C05472=1200.929,400.993,-81.846,-175.880,8.483,148.485
C05473=1200.932,400.745,-81.811,-175.880,8.481,148.484
C05474=1200.937,400.499,-81.776,-175.881,8.479,148.484
C05475=1200.941,400.250,-81.741,-175.881,8.476,148.483
C05476=1200.944,400.003,-81.706,-175.882,8.474,148.483
C05477=1200.949,399.756,-81.671,-175.882,8.471,148.482
C05478=1200.953,399.508,-81.636,-175.883,8.469,148.482
C05479=1200.957,399.261,-81.601,-175.883,8.466,148.481
C05480=1200.961,399.013,-81.566,-175.884,8.464,148.480
C05481=1200.965,398.766,-81.532,-175.884,8.462,148.480
C05482=1200.968,398.519,-81.496,-175.885,8.458,148.479
C05483=1200.972,398.270,-81.461,-175.885,8.456,148.479
C05484=1200.977,398.024,-81.426,-175.885,8.454,148.478
C05485=1200.981,397.775,-81.391,-175.886,8.451,148.478
C05486=1200.985,397.529,-81.356,-175.886,8.449,148.477
C05487=1200.989,397.281,-81.321,-175.887,8.447,148.477
C05488=1200.993,397.033,-81.287,-175.887,8.443,148.476
C05489=1200.997,396.786,-81.251,-175.888,8.441,148.476
C05490=1201.001,396.537,-81.217,-175.888,8.439,148.475
C05491=1201.004,396.291,-81.182,-175.889,8.436,148.475
C05492=1201.008,396.043,-81.147,-175.889,8.434,148.474
C05493=1201.013,395.795,-81.113,-175.890,8.430,148.473
C05494=1201.017,395.548,-81.077,-175.890,8.428,148.473
C05495=1201.021,395.301,-81.043,-175.891,8.426,148.473
C05496=1201.025,395.053,-81.007,-175.891,8.423,148.472
C05497=1201.029,394.806,-80.973,-175.892,8.421,148.471
C05498=1201.033,394.558,-80.938,-175.892,8.418,148.471
C05499=1201.036,394.310,-80.903,-175.893,8.415,148.470
C05500=1201.041,394.063,-80.868,-175.893,8.412,148.470
C05501=1201.045,393.815,-80.834,-175.894,8.410,148.469
C05502=1201.049,393.568,-80.798,-175.895,8.407,148.469
C05503=1201.053,393.320,-80.764,-175.895,8.405,148.468
C05504=1201.057,393.073,-80.730,-175.896,8.402,148.468
C05505=1201.062,392.790,-80.689,-175.896,8.400,148.467
C05506=1201.067,392.507,-80.650,-175.897,8.397,148.467
C05507=1201.070,392.224,-80.610,-175.898,8.393,148.466
C05508=1201.076,391.941,-80.570,-175.898,8.390,148.465
C05509=1201.079,391.694,-80.536,-175.899,8.387,148.465
C05510=1201.083,391.446,-80.501,-175.899,8.385,148.464
C05511=1201.088,391.199,-80.466,-175.900,8.382,148.464
C05512=1201.091,390.951,-80.431,-175.900,8.380,148.463
C05513=1201.096,390.704,-80.396,-175.901,8.376,148.463
C05514=1201.099,390.456,-80.362,-175.902,8.374,148.462
C05515=1201.104,390.209,-80.328,-175.903,8.371,148.462
C05516=1201.107,389.961,-80.292,-175.903,8.368,148.461
C05517=1201.112,389.714,-80.258,-175.904,8.365,148.460
C05518=1201.115,389.466,-80.223,-175.904,8.363,148.460
C05519=1201.120,389.218,-80.189,-175.906,8.360,148.460
C05520=1201.124,388.970,-80.154,-175.906,8.357,148.459
C05521=1201.128,388.724,-80.119,-175.907,8.355,148.458
C05522=1201.131,388.476,-80.085,-175.907,8.352,148.458
C05523=1201.136,388.228,-80.050,-175.909,8.349,148.457
C05524=1201.140,387.980,-80.015,-175.909,8.347,148.457
C05525=1201.144,387.733,-79.981,-175.910,8.343,148.456
C05526=1201.147,387.486,-79.946,-175.910,8.340,148.456
C05527=1201.152,387.238,-79.912,-175.911,8.338,148.455
C05528=1201.156,386.990,-79.877,-175.912,8.335,148.455
C05529=1201.160,386.743,-79.843,-175.913,8.332,148.454
C05530=1201.164,386.495,-79.808,-175.914,8.329,148.454
C05531=1201.168,386.247,-79.774,-175.915,8.326,148.453
C05532=1201.172,386.000,-79.740,-175.915,8.324,148.453
C05533=1201.176,385.752,-79.705,-175.916,8.321,148.452
C05534=1201.180,385.505,-79.670,-175.917,8.318,148.452
C05535=1201.184,385.257,-79.635,-175.918,8.315,148.451
C05536=1201.188,385.010,-79.601,-175.919,8.312,148.451
C05537=1201.192,384.762,-79.566,-175.920,8.309,148.450
C05538=1201.197,384.515,-79.532,-175.920,8.307,148.450
C05539=1201.200,384.267,-79.497,-175.921,8.304,148.449
C05540=1201.204,384.019,-79.463,-175.922,8.301,148.449
C05541=1201.209,383.772,-79.428,-175.923,8.298,148.448
C05542=1201.212,383.524,-79.394,-175.924,8.295,148.448
C05543=1201.217,383.277,-79.360,-175.925,8.292,148.447
C05544=1201.220,383.029,-79.326,-175.926,8.289,148.447
C05545=1201.225,382.781,-79.291,-175.927,8.286,148.446
C05546=1201.228,382.533,-79.256,-175.927,8.283,148.445
C05547=1201.232,382.286,-79.222,-175.928,8.280,148.445
C05548=1201.237,382.039,-79.188,-175.929,8.277,148.444
C05549=1201.241,381.791,-79.153,-175.930,8.275,148.444
C05550=1201.245,381.544,-79.119,-175.931,8.272,148.444
C05551=1201.249,381.295,-79.084,-175.932,8.269,148.443
C05552=1201.252,381.048,-79.051,-175.933,8.266,148.443
C05553=1201.257,380.801,-79.016,-175.934,8.263,148.442
C05554=1201.261,380.553,-78.981,-175.935,8.260,148.442
C05555=1201.265,380.306,-78.947,-175.936,8.257,148.441
C05556=1201.269,380.058,-78.913,-175.937,8.253,148.441
C05557=1201.273,379.810,-78.879,-175.938,8.251,148.440
C05558=1201.277,379.563,-78.844,-175.940,8.248,148.440
C05559=1201.281,379.315,-78.811,-175.940,8.245,148.439
C05560=1201.285,379.067,-78.776,-175.942,8.242,148.439
C05561=1201.289,378.820,-78.742,-175.942,8.239,148.438
C05562=1201.293,378.572,-78.707,-175.944,8.236,148.438
C05563=1201.298,378.325,-78.673,-175.944,8.233,148.437
C05564=1201.302,378.077,-78.639,-175.946,8.230,148.437
C05565=1201.305,377.829,-78.604,-175.947,8.227,148.436
C05566=1201.310,377.582,-78.571,-175.948,8.224,148.436
C05567=1201.314,377.334,-78.537,-175.949,8.221,148.435
C05568=1201.317,377.086,-78.502,-175.951,8.218,148.435
C05569=1201.322,376.839,-78.468,-175.951,8.215,148.434
C05570=1201.325,376.591,-78.434,-175.953,8.212,148.434
C05571=1201.330,376.343,-78.400,-175.954,8.209,148.434
C05572=1201.334,376.096,-78.366,-175.955,8.206,148.433
C05573=1201.338,375.848,-78.331,-175.956,8.203,148.433
C05574=1201.342,375.601,-78.297,-175.958,8.199,148.432
C05575=1201.346,375.354,-78.264,-175.959,8.197,148.432
C05576=1201.350,375.106,-78.230,-175.960,8.193,148.431
C05577=1201.354,374.858,-78.196,-175.961,8.191,148.431
C05578=1201.358,374.610,-78.161,-175.962,8.188,148.430
C05579=1201.362,374.363,-78.128,-175.964,8.184,148.430
C05580=1201.366,374.115,-78.093,-175.965,8.181,148.430
C05581=1201.370,373.867,-78.059,-175.966,8.178,148.429
C05582=1201.375,373.620,-78.025,-175.967,8.175,148.429
C05583=1201.378,373.372,-77.991,-175.969,8.172,148.428
C05584=1201.382,373.124,-77.957,-175.970,8.169,148.428
C05585=1201.387,372.877,-77.923,-175.971,8.166,148.427
C05586=1201.390,372.629,-77.889,-175.973,8.163,148.427
C05587=1201.395,372.381,-77.855,-175.974,8.160,148.427
C05588=1201.399,372.133,-77.822,-175.975,8.157,148.426
C05589=1201.403,371.886,-77.788,-175.976,8.154,148.426
C05590=1201.407,371.638,-77.753,-175.978,8.150,148.425
C05591=1201.411,371.391,-77.720,-175.979,8.147,148.425
C05592=1201.415,371.143,-77.686,-175.980,8.145,148.424
C05593=1201.420,370.895,-77.652,-175.982,8.141,148.424
C05594=1201.423,370.648,-77.618,-175.983,8.138,148.424
C05595=1201.427,370.400,-77.584,-175.985,8.135,148.423
C05596=1201.432,370.152,-77.550,-175.986,8.132,148.423
C05597=1201.435,369.905,-77.517,-175.988,8.129,148.422
C05598=1201.439,369.657,-77.483,-175.989,8.125,148.422
C05599=1201.443,369.409,-77.449,-175.991,8.122,148.422
C05600=1201.448,369.162,-77.415,-175.992,8.120,148.421
C05601=1201.451,368.915,-77.382,-175.994,8.116,148.421
C05602=1201.456,368.666,-77.347,-175.995,8.113,148.420
C05603=1201.460,368.419,-77.314,-175.997,8.110,148.420
C05604=1201.464,368.171,-77.280,-175.998,8.107,148.420
C05605=1201.468,367.924,-77.246,-175.999,8.104,148.419
C05606=1201.472,367.676,-77.213,-176.001,8.101,148.419
C05607=1201.476,367.427,-77.179,-176.002,8.098,148.419
C05608=1201.480,367.180,-77.145,-176.004,8.094,148.418
C05609=1201.485,366.900,-77.107,-176.006,8.091,148.418
C05610=1201.490,366.618,-77.069,-176.007,8.088,148.417
C05611=1201.494,366.338,-77.031,-176.009,8.084,148.417
C05612=1201.498,366.058,-76.993,-176.011,8.080,148.416
C05613=1201.502,365.810,-76.960,-176.012,8.077,148.416
C05614=1201.507,365.562,-76.925,-176.014,8.074,148.416
C05615=1201.511,365.315,-76.892,-176.016,8.071,148.415
C05616=1201.515,365.067,-76.859,-176.017,8.068,148.415
C05617=1201.519,364.819,-76.825,-176.019,8.064,148.414
C05618=1201.523,364.571,-76.791,-176.020,8.061,148.414
C05619=1201.527,364.324,-76.758,-176.022,8.058,148.414
C05620=1201.531,364.076,-76.724,-176.024,8.055,148.413
C05621=1201.535,363.829,-76.691,-176.025,8.052,148.413
C05622=1201.540,363.581,-76.657,-176.027,8.049,148.413
C05623=1201.543,363.332,-76.624,-176.029,8.046,148.412
C05624=1201.547,363.085,-76.590,-176.030,8.043,148.412
C05625=1201.551,362.838,-76.557,-176.032,8.039,148.412
C05626=1201.555,362.590,-76.524,-176.033,8.037,148.411
C05627=1201.560,362.342,-76.490,-176.035,8.033,148.411
C05628=1201.564,362.095,-76.456,-176.037,8.030,148.411
C05629=1201.568,361.847,-76.423,-176.039,8.027,148.410
C05630=1201.572,361.599,-76.390,-176.041,8.023,148.410
C05631=1201.576,361.351,-76.356,-176.042,8.021,148.410
C05632=1201.580,361.103,-76.323,-176.044,8.017,148.409
C05633=1201.584,360.855,-76.290,-176.046,8.014,148.409
C05634=1201.588,360.608,-76.256,-176.047,8.011,148.409
C05635=1201.592,360.361,-76.223,-176.049,8.007,148.408
C05636=1201.596,360.113,-76.190,-176.051,8.005,148.408
C05637=1201.600,359.865,-76.157,-176.053,8.001,148.408
C05638=1201.604,359.617,-76.123,-176.054,7.999,148.407
C05639=1201.609,359.369,-76.090,-176.056,7.995,148.407
C05640=1201.613,359.122,-76.057,-176.058,7.992,148.407
C05641=1201.618,358.874,-76.023,-176.060,7.989,148.407
C05642=1201.621,358.625,-75.990,-176.062,7.985,148.406
C05643=1201.625,358.378,-75.957,-176.063,7.983,148.406
C05644=1201.629,358.130,-75.924,-176.065,7.979,148.406
C05645=1201.634,357.882,-75.890,-176.067,7.976,148.405
C05646=1201.638,357.634,-75.857,-176.069,7.973,148.405
C05647=1201.642,357.387,-75.824,-176.071,7.970,148.405
C05648=1201.646,357.139,-75.791,-176.073,7.966,148.404
C05649=1201.650,356.891,-75.758,-176.074,7.964,148.404
C05650=1201.654,356.644,-75.725,-176.076,7.960,148.404
C05651=1201.658,356.396,-75.692,-176.078,7.958,148.404
C05652=1201.662,356.148,-75.659,-176.080,7.954,148.403
C05653=1201.666,355.901,-75.626,-176.082,7.951,148.403
C05654=1201.670,355.653,-75.593,-176.084,7.948,148.403
C05655=1201.674,355.405,-75.559,-176.085,7.945,148.402
C05656=1201.678,355.157,-75.526,-176.088,7.941,148.402
C05657=1201.682,354.910,-75.493,-176.089,7.939,148.402
C05658=1201.687,354.661,-75.461,-176.091,7.935,148.402
C05659=1201.691,354.414,-75.428,-176.093,7.932,148.401
C05660=1201.695,354.166,-75.394,-176.095,7.929,148.401
C05661=1201.699,353.918,-75.361,-176.097,7.926,148.401
C05662=1201.703,353.670,-75.328,-176.098,7.923,148.401
C05663=1201.707,353.423,-75.296,-176.101,7.920,148.400
C05664=1201.711,353.175,-75.263,-176.103,7.917,148.400
C05665=1201.715,352.927,-75.230,-176.104,7.914,148.400
C05666=1201.720,352.679,-75.197,-176.106,7.910,148.399
C05667=1201.724,352.432,-75.164,-176.108,7.907,148.399
C05668=1201.728,352.184,-75.130,-176.110,7.905,148.399
C05669=1201.732,351.936,-75.099,-176.112,7.901,148.399
C05670=1201.736,351.688,-75.065,-176.114,7.898,148.398
C05671=1201.740,351.440,-75.032,-176.116,7.895,148.398
C05672=1201.745,351.193,-75.000,-176.118,7.892,148.398
C05673=1201.749,350.945,-74.967,-176.120,7.888,148.398
C05674=1201.753,350.697,-74.934,-176.122,7.886,148.398
C05675=1201.757,350.449,-74.902,-176.124,7.883,148.397
C05676=1201.761,350.201,-74.869,-176.126,7.879,148.397
C05677=1201.765,349.954,-74.836,-176.128,7.876,148.397
C05678=1201.770,349.705,-74.803,-176.130,7.873,148.397
C05679=1201.773,349.458,-74.771,-176.132,7.870,148.396
C05680=1201.777,349.210,-74.738,-176.134,7.867,148.396
C05681=1201.782,348.962,-74.705,-176.136,7.864,148.396
C05682=1201.786,348.714,-74.672,-176.138,7.861,148.396
C05683=1201.790,348.467,-74.641,-176.140,7.858,148.395
C05684=1201.794,348.219,-74.607,-176.142,7.855,148.395
C05685=1201.799,347.971,-74.575,-176.144,7.851,148.395
C05686=1201.803,347.723,-74.542,-176.145,7.849,148.395
C05687=1201.806,347.476,-74.509,-176.148,7.845,148.394
C05688=1201.811,347.227,-74.477,-176.150,7.842,148.394
C05689=1201.815,346.979,-74.444,-176.152,7.839,148.394
C05690=1201.819,346.732,-74.412,-176.154,7.836,148.394
C05691=1201.823,346.484,-74.379,-176.156,7.833,148.394
C05692=1201.828,346.236,-74.347,-176.158,7.830,148.393
C05693=1201.831,345.988,-74.315,-176.160,7.827,148.393
C05694=1201.835,345.740,-74.282,-176.162,7.823,148.393
C05695=1201.840,345.492,-74.249,-176.164,7.821,148.393
C05696=1201.844,345.245,-74.217,-176.166,7.818,148.393
C05697=1201.848,344.997,-74.184,-176.168,7.814,148.392
C05698=1201.852,344.749,-74.152,-176.170,7.812,148.392
C05699=1201.856,344.501,-74.119,-176.172,7.808,148.392
C05700=1201.861,344.253,-74.087,-176.174,7.805,148.392
C05701=1201.865,344.006,-74.055,-176.176,7.803,148.392
C05702=1201.869,343.758,-74.022,-176.179,7.800,148.392
C05703=1201.873,343.510,-73.991,-176.181,7.796,148.391
C05704=1201.877,343.262,-73.957,-176.183,7.794,148.391
C05705=1201.881,343.014,-73.925,-176.185,7.790,148.391
C05706=1201.886,342.766,-73.893,-176.187,7.787,148.391
C05707=1201.890,342.519,-73.860,-176.189,7.785,148.391
C05708=1201.894,342.270,-73.828,-176.191,7.781,148.390
C05709=1201.898,342.022,-73.796,-176.193,7.778,148.390
C05710=1201.902,341.775,-73.765,-176.195,7.775,148.390
C05711=1201.906,341.527,-73.731,-176.197,7.772,148.390
C05712=1201.910,341.279,-73.700,-176.200,7.769,148.390
C05713=1201.915,341.001,-73.663,-176.202,7.766,148.389
C05714=1201.920,340.722,-73.628,-176.204,7.762,148.389
C05715=1201.924,340.443,-73.591,-176.206,7.759,148.389
C05716=1201.929,340.166,-73.555,-176.209,7.756,148.389
C05717=1201.933,339.918,-73.523,-176.211,7.753,148.389
C05718=1201.938,339.669,-73.490,-176.213,7.749,148.389
C05719=1201.942,339.422,-73.459,-176.215,7.747,148.388
C05720=1201.946,339.174,-73.427,-176.217,7.743,148.388
C05721=1201.950,338.926,-73.394,-176.220,7.740,148.388
C05722=1201.954,338.679,-73.362,-176.222,7.738,148.388
C05723=1201.959,338.430,-73.330,-176.224,7.735,148.388
C05724=1201.962,338.182,-73.298,-176.226,7.731,148.388
C05725=1201.967,337.934,-73.266,-176.228,7.729,148.387
C05726=1201.971,337.687,-73.234,-176.231,7.726,148.387
C05727=1201.975,337.439,-73.202,-176.233,7.722,148.387
C05728=1201.979,337.190,-73.170,-176.234,7.720,148.387
C05729=1201.983,336.943,-73.139,-176.237,7.716,148.387
C05730=1201.988,336.695,-73.106,-176.239,7.713,148.387
C05731=1201.992,336.447,-73.074,-176.241,7.711,148.387
C05732=1201.996,336.199,-73.043,-176.243,7.708,148.386
C05733=1202.000,335.951,-73.010,-176.245,7.704,148.386
C05734=1202.004,335.703,-72.978,-176.248,7.701,148.386
C05735=1202.008,335.456,-72.947,-176.250,7.699,148.386
C05736=1202.013,335.207,-72.915,-176.252,7.695,148.386
C05737=1202.016,334.959,-72.883,-176.255,7.692,148.386
C05738=1202.021,334.712,-72.851,-176.256,7.690,148.386
C05739=1202.025,334.463,-72.819,-176.259,7.687,148.385
C05740=1202.029,334.215,-72.787,-176.261,7.683,148.385
C05741=1202.034,333.967,-72.756,-176.263,7.681,148.385
C05742=1202.037,333.719,-72.724,-176.265,7.678,148.385
C05743=1202.042,333.472,-72.692,-176.268,7.675,148.385
C05744=1202.046,333.224,-72.660,-176.269,7.672,148.385
C05745=1202.050,332.976,-72.629,-176.272,7.669,148.385
C05746=1202.054,332.728,-72.597,-176.274,7.666,148.385
C05747=1202.059,332.479,-72.565,-176.276,7.663,148.384
C05748=1202.063,332.232,-72.534,-176.279,7.660,148.384
C05749=1202.067,331.984,-72.502,-176.281,7.657,148.384
C05750=1202.071,331.736,-72.470,-176.283,7.654,148.384
C05751=1202.075,331.489,-72.439,-176.285,7.651,148.384
C05752=1202.080,331.240,-72.407,-176.288,7.648,148.384
C05753=1202.084,330.992,-72.376,-176.290,7.645,148.384
C05754=1202.088,330.744,-72.344,-176.292,7.642,148.384
C05755=1202.092,330.496,-72.313,-176.294,7.639,148.383
C05756=1202.096,330.248,-72.281,-176.297,7.636,148.383
C05757=1202.101,330.001,-72.249,-176.298,7.634,148.383
C05758=1202.105,329.752,-72.218,-176.301,7.631,148.383
C05759=1202.109,329.505,-72.186,-176.303,7.627,148.383
C05760=1202.113,329.257,-72.155,-176.305,7.625,148.383
C05761=1202.117,329.008,-72.123,-176.308,7.622,148.383
C05762=1202.121,328.761,-72.092,-176.310,7.619,148.383
C05763=1202.125,328.513,-72.060,-176.312,7.616,148.383
C05764=1202.130,328.265,-72.029,-176.315,7.613,148.383
C05765=1202.134,328.016,-71.997,-176.317,7.610,148.382
C05766=1202.139,327.768,-71.966,-176.319,7.608,148.382
C05767=1202.142,327.520,-71.934,-176.321,7.604,148.382
C05768=1202.147,327.272,-71.903,-176.324,7.601,148.382
C05769=1202.151,327.024,-71.872,-176.326,7.598,148.382
C05770=1202.155,326.777,-71.840,-176.328,7.596,148.382
C05771=1202.159,326.528,-71.809,-176.331,7.592,148.382
C05772=1202.163,326.281,-71.778,-176.333,7.589,148.382
C05773=1202.167,326.032,-71.746,-176.335,7.587,148.382
C05774=1202.172,325.785,-71.715,-176.338,7.584,148.382
C05775=1202.176,325.537,-71.684,-176.340,7.580,148.381
C05776=1202.180,325.288,-71.653,-176.342,7.578,148.382
C05777=1202.185,325.041,-71.622,-176.344,7.575,148.381
C05778=1202.189,324.792,-71.590,-176.347,7.572,148.381
C05779=1202.193,324.545,-71.559,-176.349,7.570,148.381
C05780=1202.197,324.296,-71.528,-176.351,7.566,148.381
C05781=1202.201,324.049,-71.496,-176.354,7.563,148.381
C05782=1202.205,323.800,-71.465,-176.356,7.561,148.381
C05783=1202.210,323.552,-71.434,-176.358,7.558,148.381
C05784=1202.214,323.304,-71.403,-176.360,7.554,148.381
C05785=1202.218,323.056,-71.372,-176.363,7.552,148.381
C05786=1202.223,322.808,-71.341,-176.365,7.549,148.381
C05787=1202.226,322.560,-71.309,-176.367,7.546,148.381
C05788=1202.230,322.313,-71.279,-176.370,7.544,148.381
C05789=1202.234,322.064,-71.248,-176.372,7.540,148.380
C05790=1202.239,321.816,-71.217,-176.375,7.537,148.380
C05791=1202.243,321.569,-71.186,-176.377,7.534,148.380
C05792=1202.247,321.320,-71.155,-176.379,7.532,148.380
C05793=1202.252,321.072,-71.124,-176.382,7.529,148.380
C05794=1202.256,320.823,-71.093,-176.384,7.526,148.380
C05795=1202.260,320.576,-71.061,-176.386,7.523,148.380
C05796=1202.264,320.329,-71.031,-176.389,7.520,148.380
C05797=1202.268,320.080,-71.000,-176.391,7.517,148.380
C05798=1202.273,319.832,-70.969,-176.393,7.515,148.380
C05799=1202.277,319.584,-70.938,-176.396,7.512,148.380
C05800=1202.281,319.336,-70.907,-176.398,7.509,148.380
C05801=1202.286,319.088,-70.876,-176.400,7.506,148.380
C05802=1202.290,318.840,-70.846,-176.403,7.503,148.380
C05803=1202.294,318.592,-70.814,-176.405,7.500,148.380
C05804=1202.298,318.344,-70.784,-176.407,7.498,148.380
C05805=1202.303,318.096,-70.753,-176.410,7.495,148.380
C05806=1202.307,317.847,-70.722,-176.412,7.491,148.380
C05807=1202.311,317.599,-70.692,-176.414,7.489,148.380
C05808=1202.315,317.351,-70.661,-176.417,7.486,148.380
C05809=1202.319,317.103,-70.630,-176.419,7.483,148.380
C05810=1202.324,316.855,-70.599,-176.422,7.481,148.380
C05811=1202.327,316.608,-70.568,-176.424,7.477,148.379
C05812=1202.331,316.359,-70.537,-176.426,7.474,148.379
C05813=1202.336,316.111,-70.506,-176.429,7.472,148.379
C05814=1202.340,315.863,-70.477,-176.431,7.469,148.379
C05815=1202.345,315.615,-70.446,-176.434,7.466,148.379
C05816=1202.349,315.366,-70.415,-176.436,7.464,148.379
C05817=1202.354,315.091,-70.381,-176.438,7.461,148.379
C05818=1202.358,314.815,-70.346,-176.441,7.458,148.379
C05819=1202.364,314.538,-70.313,-176.444,7.455,148.379
C05820=1202.368,314.262,-70.278,-176.446,7.450,148.379
C05821=1202.372,314.014,-70.248,-176.449,7.448,148.379
C05822=1202.376,313.766,-70.217,-176.451,7.445,148.379
C05823=1202.381,313.518,-70.187,-176.454,7.442,148.379
C05824=1202.384,313.269,-70.157,-176.456,7.440,148.379
C05825=1202.389,313.021,-70.126,-176.458,7.437,148.379
C05826=1202.393,312.774,-70.096,-176.461,7.434,148.379
C05827=1202.398,312.526,-70.065,-176.463,7.431,148.379
C05828=1202.402,312.277,-70.034,-176.466,7.428,148.379
C05829=1202.406,312.029,-70.004,-176.468,7.426,148.379
C05830=1202.410,311.781,-69.974,-176.470,7.423,148.379
C05831=1202.414,311.533,-69.943,-176.473,7.420,148.379
C05832=1202.419,311.285,-69.913,-176.475,7.418,148.379
C05833=1202.423,311.036,-69.882,-176.478,7.415,148.379
C05834=1202.427,310.788,-69.852,-176.480,7.412,148.379
C05835=1202.432,310.540,-69.821,-176.482,7.409,148.379
C05836=1202.435,310.293,-69.791,-176.485,7.406,148.379
C05837=1202.440,310.044,-69.761,-176.487,7.403,148.379
C05838=1202.444,309.796,-69.731,-176.490,7.401,148.379
C05839=1202.448,309.548,-69.700,-176.492,7.398,148.379
C05840=1202.452,309.300,-69.670,-176.495,7.395,148.379
C05841=1202.457,309.052,-69.640,-176.497,7.392,148.379
C05842=1202.461,308.804,-69.609,-176.499,7.389,148.379
C05843=1202.466,308.555,-69.579,-176.502,7.386,148.379
C05844=1202.470,308.308,-69.549,-176.504,7.384,148.379
C05845=1202.475,308.059,-69.519,-176.507,7.381,148.379
C05846=1202.479,307.811,-69.489,-176.509,7.379,148.379
C05847=1202.483,307.563,-69.458,-176.512,7.376,148.379
C05848=1202.487,307.315,-69.428,-176.514,7.373,148.379
C05849=1202.491,307.067,-69.398,-176.516,7.370,148.379
C05850=1202.496,306.818,-69.368,-176.519,7.367,148.379
C05851=1202.499,306.571,-69.338,-176.521,7.364,148.379
C05852=1202.504,306.322,-69.308,-176.523,7.362,148.379
C05853=1202.508,306.074,-69.278,-176.526,7.359,148.379
C05854=1202.513,305.826,-69.248,-176.529,7.356,148.379
C05855=1202.517,305.578,-69.218,-176.531,7.354,148.379
C05856=1202.521,305.330,-69.188,-176.534,7.351,148.379
C05857=1202.526,305.081,-69.158,-176.536,7.349,148.379
C05858=1202.529,304.833,-69.127,-176.539,7.346,148.379
C05859=1202.534,304.585,-69.098,-176.541,7.342,148.379
C05860=1202.538,304.337,-69.067,-176.543,7.340,148.379
C05861=1202.542,304.089,-69.038,-176.546,7.337,148.379
C05862=1202.546,303.841,-69.008,-176.548,7.334,148.379
C05863=1202.551,303.592,-68.978,-176.550,7.332,148.379
C05864=1202.555,303.344,-68.948,-176.553,7.329,148.379
C05865=1202.559,303.096,-68.918,-176.555,7.327,148.379
C05866=1202.564,302.848,-68.888,-176.558,7.324,148.379
C05867=1202.568,302.600,-68.858,-176.561,7.320,148.379
C05868=1202.572,302.352,-68.828,-176.563,7.318,148.379
C05869=1202.577,302.103,-68.798,-176.565,7.315,148.379
C05870=1202.581,301.855,-68.769,-176.568,7.313,148.379
C05871=1202.585,301.607,-68.739,-176.570,7.310,148.379
C05872=1202.589,301.359,-68.709,-176.573,7.307,148.379
C05873=1202.594,301.111,-68.679,-176.575,7.305,148.379
C05874=1202.598,300.862,-68.650,-176.578,7.302,148.379
C05875=1202.603,300.614,-68.620,-176.580,7.299,148.379
C05876=1202.606,300.366,-68.590,-176.583,7.297,148.379
C05877=1202.611,300.118,-68.561,-176.585,7.294,148.379
C05878=1202.616,299.870,-68.531,-176.587,7.291,148.379
C05879=1202.620,299.621,-68.501,-176.590,7.288,148.379
C05880=1202.624,299.373,-68.472,-176.593,7.285,148.379
C05881=1202.628,299.125,-68.442,-176.595,7.283,148.380
C05882=1202.632,298.877,-68.412,-176.598,7.280,148.380
C05883=1202.637,298.629,-68.382,-176.600,7.278,148.380
C05884=1202.641,298.380,-68.353,-176.602,7.275,148.380
C05885=1202.646,298.133,-68.323,-176.605,7.272,148.380
C05886=1202.650,297.884,-68.294,-176.607,7.270,148.380
C05887=1202.654,297.636,-68.265,-176.610,7.267,148.380
C05888=1202.658,297.388,-68.235,-176.612,7.265,148.380
C05889=1202.663,297.140,-68.206,-176.615,7.261,148.380
C05890=1202.667,296.891,-68.176,-176.617,7.258,148.380
C05891=1202.671,296.643,-68.147,-176.620,7.256,148.380
C05892=1202.676,296.394,-68.117,-176.622,7.253,148.380
C05893=1202.680,296.146,-68.087,-176.624,7.251,148.380
C05894=1202.684,295.898,-68.058,-176.627,7.248,148.380
C05895=1202.688,295.650,-68.028,-176.629,7.246,148.380
C05896=1202.693,295.401,-67.999,-176.632,7.243,148.380
C05897=1202.697,295.154,-67.970,-176.635,7.240,148.380
C05898=1202.702,294.906,-67.940,-176.637,7.238,148.380
C05899=1202.706,294.657,-67.911,-176.640,7.235,148.380
C05900=1202.710,294.409,-67.881,-176.642,7.233,148.380
C05901=1202.714,294.161,-67.852,-176.645,7.230,148.380
C05902=1202.718,293.913,-67.822,-176.647,7.227,148.380
C05903=1202.723,293.664,-67.793,-176.650,7.225,148.381
C05904=1202.728,293.416,-67.765,-176.652,7.221,148.381
C05905=1202.732,293.168,-67.735,-176.654,7.219,148.381
C05906=1202.736,292.920,-67.706,-176.657,7.216,148.381
C05907=1202.740,292.671,-67.676,-176.659,7.214,148.381
C05908=1202.744,292.423,-67.647,-176.662,7.211,148.381
C05909=1202.749,292.175,-67.617,-176.665,7.208,148.381
C05910=1202.754,291.927,-67.589,-176.667,7.206,148.381
C05911=1202.758,291.678,-67.560,-176.670,7.203,148.381
C05912=1202.762,291.430,-67.530,-176.672,7.201,148.381
C05913=1202.765,291.182,-67.501,-176.675,7.198,148.381
C05914=1202.770,290.933,-67.473,-176.677,7.196,148.381
C05915=1202.774,290.685,-67.443,-176.680,7.193,148.381
C05916=1202.779,290.437,-67.414,-176.682,7.191,148.381
C05917=1202.783,290.189,-67.385,-176.684,7.188,148.381
C05918=1202.788,289.940,-67.356,-176.688,7.185,148.382
C05919=1202.792,289.692,-67.326,-176.690,7.183,148.382
C05920=1202.796,289.444,-67.297,-176.692,7.180,148.382
C05921=1202.801,289.169,-67.265,-176.695,7.177,148.382
C05922=1202.805,288.895,-67.234,-176.697,7.174,148.382
C05923=1202.810,288.621,-67.201,-176.700,7.172,148.382
C05924=1202.816,288.347,-67.169,-176.703,7.169,148.382
C05925=1202.819,288.098,-67.141,-176.706,7.166,148.382
C05926=1202.823,287.850,-67.111,-176.708,7.163,148.382
C05927=1202.828,287.602,-67.082,-176.711,7.160,148.382
C05928=1202.833,287.353,-67.054,-176.713,7.159,148.382
C05929=1202.837,287.105,-67.024,-176.716,7.156,148.382
C05930=1202.841,286.857,-66.996,-176.719,7.153,148.383
C05931=1202.845,286.609,-66.967,-176.721,7.150,148.383
C05932=1202.850,286.360,-66.938,-176.723,7.147,148.383
C05933=1202.854,286.112,-66.909,-176.726,7.145,148.383
C05934=1202.858,285.864,-66.881,-176.729,7.142,148.383
C05935=1202.863,285.616,-66.851,-176.731,7.140,148.383
C05936=1202.867,285.367,-66.823,-176.734,7.137,148.383
C05937=1202.872,285.119,-66.794,-176.736,7.135,148.383
C05938=1202.876,284.870,-66.766,-176.738,7.132,148.383
C05939=1202.880,284.622,-66.736,-176.741,7.130,148.383
C05940=1202.885,284.374,-66.708,-176.744,7.127,148.383
C05941=1202.889,284.125,-66.680,-176.746,7.125,148.383
C05942=1202.893,283.877,-66.650,-176.749,7.122,148.384
C05943=1202.898,283.629,-66.622,-176.751,7.120,148.384
C05944=1202.902,283.381,-66.592,-176.754,7.117,148.384
C05945=1202.906,283.132,-66.564,-176.756,7.115,148.384
C05946=1202.911,282.884,-66.536,-176.759,7.112,148.384
C05947=1202.915,282.636,-66.506,-176.761,7.110,148.384
C05948=1202.919,282.387,-66.478,-176.764,7.107,148.384
C05949=1202.924,282.139,-66.450,-176.766,7.105,148.384
C05950=1202.927,281.891,-66.421,-176.769,7.102,148.384
C05951=1202.933,281.643,-66.393,-176.771,7.100,148.384
C05952=1202.937,281.394,-66.364,-176.774,7.097,148.384
C05953=1202.941,281.145,-66.336,-176.776,7.094,148.385
C05954=1202.946,280.898,-66.307,-176.779,7.092,148.385
C05955=1202.949,280.649,-66.278,-176.781,7.090,148.385
C05956=1202.954,280.401,-66.250,-176.784,7.087,148.385
C05957=1202.959,280.152,-66.221,-176.786,7.084,148.385
C05958=1202.963,279.904,-66.193,-176.789,7.082,148.385
C05959=1202.967,279.656,-66.164,-176.791,7.079,148.385
C05960=1202.971,279.407,-66.136,-176.794,7.076,148.385
C05961=1202.976,279.159,-66.108,-176.796,7.074,148.385
C05962=1202.980,278.911,-66.079,-176.799,7.072,148.386
C05963=1202.984,278.662,-66.051,-176.801,7.069,148.386
C05964=1202.989,278.414,-66.023,-176.804,7.066,148.386
C05965=1202.993,278.166,-65.993,-176.806,7.064,148.386
C05966=1202.997,277.918,-65.966,-176.809,7.061,148.386
C05967=1203.002,277.669,-65.937,-176.812,7.059,148.386
C05968=1203.006,277.421,-65.909,-176.814,7.056,148.386
C05969=1203.011,277.172,-65.880,-176.817,7.054,148.386
C05970=1203.015,276.924,-65.853,-176.820,7.051,148.387
C05971=1203.020,276.675,-65.824,-176.822,7.049,148.387
C05972=1203.024,276.427,-65.796,-176.824,7.046,148.387
C05973=1203.028,276.179,-65.768,-176.827,7.044,148.387
C05974=1203.033,275.931,-65.740,-176.830,7.041,148.387
C05975=1203.036,275.682,-65.711,-176.832,7.039,148.387
C05976=1203.042,275.434,-65.683,-176.835,7.036,148.387
C05977=1203.045,275.185,-65.655,-176.837,7.034,148.387
C05978=1203.050,274.937,-65.627,-176.839,7.032,148.387
C05979=1203.054,274.689,-65.598,-176.842,7.029,148.387
C05980=1203.058,274.441,-65.571,-176.845,7.027,148.388
C05981=1203.063,274.192,-65.542,-176.847,7.024,148.388
C05982=1203.067,273.944,-65.514,-176.850,7.022,148.388
C05983=1203.071,273.695,-65.486,-176.853,7.019,148.388
C05984=1203.076,273.447,-65.458,-176.855,7.017,148.388
C05985=1203.080,273.198,-65.430,-176.858,7.014,148.388
C05986=1203.085,272.950,-65.402,-176.860,7.012,148.389
C05987=1203.089,272.701,-65.374,-176.863,7.009,148.389
C05988=1203.093,272.453,-65.346,-176.865,7.007,148.389
C05989=1203.097,272.205,-65.318,-176.868,7.005,148.389
C05990=1203.103,271.956,-65.290,-176.870,7.002,148.389
C05991=1203.107,271.708,-65.262,-176.872,7.000,148.389
C05992=1203.111,271.459,-65.234,-176.876,6.997,148.389
C05993=1203.116,271.211,-65.206,-176.878,6.995,148.389
C05994=1203.120,270.963,-65.178,-176.880,6.992,148.389
C05995=1203.124,270.714,-65.151,-176.883,6.990,148.390
C05996=1203.129,270.466,-65.123,-176.885,6.988,148.390
C05997=1203.133,270.217,-65.094,-176.888,6.985,148.390
C05998=1203.137,269.970,-65.066,-176.891,6.983,148.390
C05999=1203.141,269.720,-65.039,-176.893,6.980,148.390
C06000=1203.146,269.473,-65.011,-176.895,6.978,148.390
C06001=1203.151,269.224,-64.983,-176.899,6.975,148.391
C06002=1203.155,268.975,-64.955,-176.901,6.973,148.391
C06003=1203.159,268.727,-64.928,-176.903,6.971,148.391
C06004=1203.164,268.479,-64.900,-176.906,6.968,148.391
C06005=1203.168,268.230,-64.872,-176.908,6.966,148.391
C06006=1203.173,267.982,-64.844,-176.911,6.963,148.391
C06007=1203.177,267.733,-64.817,-176.914,6.961,148.391
C06008=1203.181,267.485,-64.789,-176.916,6.958,148.391
C06009=1203.186,267.237,-64.761,-176.919,6.956,148.392
C06010=1203.190,266.988,-64.734,-176.921,6.954,148.392
C06011=1203.194,266.740,-64.706,-176.924,6.951,148.392
C06012=1203.199,266.491,-64.678,-176.926,6.949,148.392
C06013=1203.203,266.243,-64.650,-176.929,6.946,148.392
C06014=1203.208,265.994,-64.623,-176.932,6.944,148.392
C06015=1203.212,265.746,-64.595,-176.934,6.942,148.393
C06016=1203.217,265.498,-64.568,-176.936,6.939,148.393
C06017=1203.220,265.249,-64.540,-176.939,6.937,148.393
C06018=1203.225,265.001,-64.513,-176.942,6.934,148.393
C06019=1203.229,264.753,-64.485,-176.944,6.932,148.393
C06020=1203.234,264.504,-64.458,-176.947,6.930,148.393
C06021=1203.238,264.256,-64.430,-176.949,6.927,148.393
C06022=1203.243,264.007,-64.402,-176.952,6.925,148.394
C06023=1203.248,263.758,-64.375,-176.954,6.923,148.394
C06024=1203.252,263.510,-64.347,-176.957,6.920,148.394
C06025=1203.256,263.238,-64.317,-176.960,6.918,148.394
C06026=1203.261,262.965,-64.287,-176.963,6.916,148.394
C06027=1203.265,262.692,-64.257,-176.965,6.913,148.394
C06028=1203.271,262.419,-64.227,-176.968,6.910,148.395
C06029=1203.275,262.171,-64.200,-176.971,6.908,148.395
C06030=1203.280,261.922,-64.173,-176.973,6.906,148.395
C06031=1203.284,261.673,-64.145,-176.976,6.903,148.395
C06032=1203.288,261.425,-64.117,-176.978,6.901,148.395
C06033=1203.293,261.177,-64.090,-176.981,6.898,148.395
C06034=1203.298,260.928,-64.063,-176.983,6.896,148.396
C06035=1203.301,260.680,-64.035,-176.986,6.894,148.396
C06036=1203.306,260.431,-64.008,-176.989,6.891,148.396
C06037=1203.311,260.183,-63.981,-176.991,6.889,148.396
C06038=1203.315,259.934,-63.954,-176.993,6.887,148.396
C06039=1203.320,259.686,-63.926,-176.996,6.884,148.396
C06040=1203.324,259.437,-63.899,-176.999,6.882,148.397
C06041=1203.328,259.189,-63.872,-177.001,6.880,148.397
C06042=1203.332,258.940,-63.845,-177.004,6.877,148.397
C06043=1203.337,258.692,-63.818,-177.006,6.875,148.397
C06044=1203.341,258.444,-63.790,-177.009,6.873,148.397
C06045=1203.346,258.196,-63.763,-177.012,6.870,148.397
C06046=1203.350,257.946,-63.736,-177.014,6.868,148.398
C06047=1203.355,257.698,-63.709,-177.016,6.866,148.398
C06048=1203.359,257.449,-63.682,-177.020,6.864,148.398
C06049=1203.363,257.201,-63.655,-177.022,6.861,148.398
C06050=1203.368,256.953,-63.628,-177.024,6.859,148.398
C06051=1203.373,256.704,-63.601,-177.027,6.856,148.398
C06052=1203.377,256.455,-63.574,-177.029,6.854,148.399
C06053=1203.381,256.206,-63.547,-177.032,6.852,148.399
C06054=1203.386,255.958,-63.520,-177.034,6.849,148.399
C06055=1203.390,255.710,-63.492,-177.037,6.848,148.399
C06056=1203.394,255.462,-63.465,-177.039,6.845,148.399
C06057=1203.399,255.213,-63.438,-177.042,6.843,148.400
C06058=1203.404,254.965,-63.411,-177.045,6.841,148.400
C06059=1203.408,254.717,-63.385,-177.047,6.839,148.400
C06060=1203.412,254.468,-63.358,-177.050,6.836,148.400
C06061=1203.417,254.218,-63.331,-177.053,6.834,148.400
C06062=1203.421,253.970,-63.304,-177.055,6.832,148.400
C06063=1203.425,253.722,-63.277,-177.058,6.829,148.401
C06064=1203.430,253.473,-63.250,-177.060,6.827,148.401
C06065=1203.434,253.225,-63.223,-177.063,6.825,148.401
C06066=1203.439,252.976,-63.196,-177.065,6.822,148.401
C06067=1203.443,252.728,-63.170,-177.068,6.820,148.401
C06068=1203.448,252.480,-63.143,-177.070,6.818,148.402
C06069=1203.452,252.231,-63.116,-177.073,6.815,148.402
C06070=1203.456,251.983,-63.089,-177.075,6.813,148.402
C06071=1203.461,251.734,-63.063,-177.078,6.811,148.402
C06072=1203.466,251.485,-63.036,-177.080,6.809,148.402
C06073=1203.470,251.237,-63.009,-177.083,6.806,148.403
C06074=1203.474,250.989,-62.982,-177.086,6.804,148.403
C06075=1203.479,250.740,-62.955,-177.088,6.802,148.403
C06076=1203.483,250.491,-62.929,-177.091,6.800,148.403
C06077=1203.488,250.243,-62.902,-177.094,6.797,148.403
C06078=1203.492,249.995,-62.876,-177.096,6.796,148.404
C06079=1203.497,249.746,-62.849,-177.098,6.793,148.404
C06080=1203.501,249.498,-62.822,-177.101,6.791,148.404
C06081=1203.505,249.249,-62.796,-177.104,6.789,148.404
C06082=1203.510,249.000,-62.769,-177.106,6.787,148.404
C06083=1203.514,248.752,-62.742,-177.109,6.784,148.405
C06084=1203.519,248.503,-62.716,-177.112,6.782,148.405
C06085=1203.524,248.255,-62.689,-177.114,6.780,148.405
C06086=1203.528,248.006,-62.663,-177.116,6.778,148.405
C06087=1203.533,247.757,-62.636,-177.120,6.775,148.405
C06088=1203.536,247.509,-62.610,-177.122,6.773,148.406
C06089=1203.541,247.261,-62.583,-177.124,6.771,148.406
C06090=1203.545,247.012,-62.557,-177.127,6.768,148.406
C06091=1203.550,246.763,-62.530,-177.130,6.766,148.406
C06092=1203.554,246.514,-62.504,-177.132,6.764,148.406
C06093=1203.559,246.266,-62.477,-177.134,6.762,148.407
C06094=1203.563,246.018,-62.451,-177.137,6.759,148.407
C06095=1203.568,245.769,-62.424,-177.140,6.757,148.407
C06096=1203.572,245.520,-62.398,-177.142,6.756,148.407
C06097=1203.577,245.271,-62.372,-177.145,6.753,148.407
C06098=1203.581,245.023,-62.345,-177.148,6.751,148.408
C06099=1203.585,244.774,-62.319,-177.150,6.749,148.408
C06100=1203.589,244.526,-62.292,-177.153,6.747,148.408
C06101=1203.595,244.277,-62.266,-177.155,6.745,148.408
C06102=1203.599,244.029,-62.240,-177.158,6.742,148.409
C06103=1203.603,243.780,-62.214,-177.161,6.740,148.409
C06104=1203.608,243.532,-62.187,-177.163,6.738,148.409
C06105=1203.612,243.283,-62.161,-177.165,6.736,148.409
C06106=1203.617,243.035,-62.134,-177.168,6.733,148.409
C06107=1203.621,242.786,-62.108,-177.171,6.731,148.410
C06108=1203.625,242.537,-62.083,-177.173,6.729,148.410
C06109=1203.630,242.289,-62.056,-177.175,6.727,148.410
C06110=1203.635,242.040,-62.030,-177.179,6.724,148.410
C06111=1203.639,241.792,-62.003,-177.181,6.722,148.410
C06112=1203.643,241.543,-61.977,-177.183,6.720,148.411
C06113=1203.648,241.294,-61.952,-177.186,6.719,148.411
C06114=1203.652,241.046,-61.925,-177.188,6.716,148.411
C06115=1203.657,240.797,-61.899,-177.191,6.714,148.411
C06116=1203.661,240.548,-61.873,-177.194,6.712,148.412
C06117=1203.666,240.300,-61.846,-177.196,6.710,148.412
C06118=1203.670,240.052,-61.821,-177.199,6.708,148.412
C06119=1203.675,239.803,-61.795,-177.201,6.705,148.412
C06120=1203.679,239.554,-61.768,-177.204,6.703,148.413
C06121=1203.683,239.306,-61.742,-177.207,6.701,148.413
C06122=1203.688,239.057,-61.717,-177.209,6.699,148.413
C06123=1203.692,238.809,-61.691,-177.212,6.697,148.413
C06124=1203.697,238.560,-61.664,-177.215,6.694,148.414
C06125=1203.701,238.311,-61.638,-177.217,6.692,148.414
C06126=1203.706,238.063,-61.612,-177.220,6.690,148.414
C06127=1203.710,237.814,-61.587,-177.222,6.688,148.414
C06128=1203.715,237.565,-61.561,-177.224,6.686,148.414
C06129=1203.720,237.294,-61.532,-177.227,6.684,148.415
C06130=1203.724,237.022,-61.504,-177.230,6.682,148.415
C06131=1203.729,236.752,-61.475,-177.233,6.679,148.415
C06132=1203.734,236.480,-61.447,-177.235,6.677,148.415
C06133=1203.738,236.231,-61.422,-177.239,6.674,148.416
C06134=1203.744,235.982,-61.396,-177.241,6.673,148.416
C06135=1203.748,235.734,-61.370,-177.243,6.670,148.416
C06136=1203.752,235.485,-61.344,-177.246,6.669,148.416
C06137=1203.757,235.236,-61.318,-177.249,6.667,148.417
C06138=1203.761,234.988,-61.293,-177.251,6.664,148.417
C06139=1203.766,234.739,-61.267,-177.254,6.662,148.417
C06140=1203.770,234.491,-61.240,-177.257,6.660,148.417
C06141=1203.775,234.243,-61.215,-177.259,6.658,148.418
C06142=1203.779,233.994,-61.189,-177.261,6.656,148.418
C06143=1203.784,233.745,-61.163,-177.265,6.653,148.418
C06144=1203.788,233.496,-61.138,-177.267,6.651,148.418
C06145=1203.793,233.248,-61.112,-177.269,6.649,148.419
C06146=1203.797,232.999,-61.086,-177.272,6.647,148.419
C06147=1203.801,232.750,-61.061,-177.274,6.645,148.419
C06148=1203.806,232.502,-61.036,-177.277,6.643,148.419
C06149=1203.811,232.253,-61.010,-177.280,6.641,148.420
C06150=1203.815,232.004,-60.984,-177.282,6.639,148.420
C06151=1203.820,231.756,-60.959,-177.285,6.637,148.420
C06152=1203.824,231.507,-60.933,-177.288,6.635,148.420
C06153=1203.829,231.258,-60.907,-177.290,6.633,148.420
C06154=1203.833,231.010,-60.882,-177.292,6.631,148.421
C06155=1203.838,230.761,-60.856,-177.295,6.628,148.421
C06156=1203.842,230.512,-60.830,-177.298,6.626,148.421
C06157=1203.847,230.264,-60.806,-177.300,6.624,148.421
C06158=1203.851,230.015,-60.780,-177.303,6.622,148.422
C06159=1203.855,229.766,-60.754,-177.306,6.621,148.422
C06160=1203.860,229.518,-60.729,-177.308,6.618,148.422
C06161=1203.865,229.269,-60.703,-177.311,6.616,148.423
C06162=1203.869,229.021,-60.677,-177.314,6.614,148.423
C06163=1203.874,228.772,-60.652,-177.316,6.612,148.423
C06164=1203.878,228.523,-60.627,-177.318,6.610,148.423
C06165=1203.883,228.275,-60.601,-177.321,6.608,148.424
C06166=1203.887,228.026,-60.576,-177.324,6.606,148.424
C06167=1203.892,227.777,-60.551,-177.326,6.603,148.424
C06168=1203.897,227.528,-60.525,-177.329,6.601,148.424
C06169=1203.900,227.280,-60.500,-177.332,6.600,148.425
C06170=1203.905,227.031,-60.475,-177.334,6.598,148.425
C06171=1203.909,226.782,-60.450,-177.336,6.596,148.425
C06172=1203.914,226.534,-60.424,-177.339,6.594,148.425
C06173=1203.919,226.285,-60.399,-177.342,6.592,148.426
C06174=1203.923,226.036,-60.373,-177.345,6.589,148.426
C06175=1203.928,225.788,-60.348,-177.347,6.587,148.426
C06176=1203.932,225.538,-60.323,-177.350,6.585,148.426
C06177=1203.937,225.290,-60.298,-177.352,6.583,148.427
C06178=1203.941,225.042,-60.272,-177.355,6.582,148.427
C06179=1203.946,224.793,-60.248,-177.357,6.579,148.427
C06180=1203.950,224.544,-60.222,-177.360,6.578,148.428
C06181=1203.955,224.296,-60.197,-177.362,6.576,148.428
C06182=1203.959,224.047,-60.172,-177.366,6.573,148.428
C06183=1203.964,223.798,-60.147,-177.368,6.571,148.428
C06184=1203.968,223.550,-60.122,-177.370,6.569,148.429
C06185=1203.973,223.301,-60.096,-177.373,6.567,148.429
C06186=1203.977,223.052,-60.071,-177.376,6.565,148.429
C06187=1203.982,222.804,-60.046,-177.378,6.564,148.430
C06188=1203.987,222.555,-60.021,-177.380,6.561,148.430
C06189=1203.991,222.307,-59.996,-177.383,6.560,148.430
C06190=1203.995,222.057,-59.971,-177.386,6.557,148.430
C06191=1204.000,221.809,-59.946,-177.389,6.555,148.431
C06192=1204.005,221.560,-59.921,-177.391,6.553,148.431
C06193=1204.009,221.311,-59.897,-177.394,6.551,148.431
C06194=1204.013,221.063,-59.871,-177.396,6.549,148.431
C06195=1204.018,220.814,-59.846,-177.399,6.547,148.432
C06196=1204.022,220.565,-59.821,-177.402,6.546,148.432
C06197=1204.027,220.317,-59.796,-177.404,6.543,148.432
C06198=1204.032,220.067,-59.771,-177.406,6.542,148.433
C06199=1204.036,219.819,-59.746,-177.410,6.539,148.433
C06200=1204.040,219.570,-59.721,-177.412,6.537,148.433
C06201=1204.045,219.321,-59.697,-177.415,6.535,148.433
C06202=1204.050,219.073,-59.671,-177.417,6.533,148.434
C06203=1204.054,218.824,-59.647,-177.420,6.531,148.434
C06204=1204.059,218.575,-59.622,-177.422,6.529,148.434
C06205=1204.063,218.326,-59.597,-177.425,6.528,148.435
C06206=1204.068,218.078,-59.573,-177.428,6.526,148.435
C06207=1204.072,217.829,-59.547,-177.430,6.524,148.435
C06208=1204.076,217.581,-59.523,-177.433,6.521,148.435
C06209=1204.081,217.332,-59.498,-177.436,6.519,148.436
C06210=1204.086,217.083,-59.473,-177.438,6.517,148.436
C06211=1204.090,216.834,-59.449,-177.441,6.515,148.436
C06212=1204.095,216.585,-59.424,-177.444,6.514,148.437
C06213=1204.100,216.337,-59.398,-177.446,6.511,148.437
C06214=1204.104,216.088,-59.374,-177.448,6.510,148.437
C06215=1204.109,215.839,-59.349,-177.451,6.508,148.437
C06216=1204.113,215.591,-59.325,-177.454,6.506,148.438
C06217=1204.118,215.342,-59.301,-177.456,6.504,148.438
C06218=1204.122,215.093,-59.275,-177.459,6.502,148.438
C06219=1204.127,214.845,-59.251,-177.462,6.499,148.439
C06220=1204.131,214.595,-59.226,-177.464,6.497,148.439
C06221=1204.136,214.347,-59.202,-177.467,6.496,148.439
C06222=1204.140,214.098,-59.178,-177.470,6.494,148.440
C06223=1204.145,213.849,-59.153,-177.472,6.492,148.440
C06224=1204.150,213.600,-59.128,-177.475,6.490,148.440
C06225=1204.154,213.352,-59.104,-177.477,6.488,148.440
C06226=1204.159,213.102,-59.079,-177.480,6.486,148.441
C06227=1204.163,212.854,-59.055,-177.482,6.484,148.441
C06228=1204.167,212.606,-59.030,-177.485,6.482,148.441
C06229=1204.172,212.357,-59.005,-177.488,6.481,148.442
C06230=1204.176,212.108,-58.981,-177.490,6.479,148.442
C06231=1204.181,211.860,-58.956,-177.493,6.477,148.442
C06232=1204.186,211.611,-58.932,-177.496,6.474,148.442
C06233=1204.190,211.340,-58.906,-177.498,6.472,148.443
C06234=1204.196,211.070,-58.879,-177.501,6.471,148.443
C06235=1204.201,210.799,-58.852,-177.504,6.469,148.444
C06236=1204.206,210.529,-58.826,-177.507,6.466,148.444
C06237=1204.210,210.280,-58.801,-177.509,6.464,148.444
C06238=1204.214,210.032,-58.777,-177.512,6.462,148.444
C06239=1204.220,209.782,-58.753,-177.515,6.460,148.445
C06240=1204.224,209.534,-58.729,-177.517,6.458,148.445
C06241=1204.228,209.284,-58.704,-177.520,6.457,148.445
C06242=1204.233,209.036,-58.680,-177.523,6.455,148.446
C06243=1204.237,208.788,-58.656,-177.525,6.453,148.446
C06244=1204.242,208.539,-58.631,-177.528,6.451,148.446
C06245=1204.246,208.290,-58.607,-177.530,6.449,148.447
C06246=1204.251,208.041,-58.583,-177.533,6.447,148.447
C06247=1204.256,207.792,-58.559,-177.535,6.445,148.447
C06248=1204.260,207.544,-58.535,-177.538,6.444,148.448
C06249=1204.265,207.295,-58.511,-177.541,6.442,148.448
C06250=1204.269,207.046,-58.486,-177.543,6.440,148.448
C06251=1204.274,206.797,-58.461,-177.546,6.438,148.449
C06252=1204.278,206.548,-58.438,-177.549,6.436,148.449
C06253=1204.284,206.300,-58.413,-177.552,6.434,148.449
C06254=1204.288,206.051,-58.389,-177.555,6.432,148.450
C06255=1204.292,205.802,-58.365,-177.557,6.430,148.450
C06256=1204.296,205.553,-58.342,-177.559,6.428,148.450
C06257=1204.302,205.304,-58.317,-177.562,6.426,148.450
C06258=1204.306,205.056,-58.293,-177.565,6.424,148.451
C06259=1204.311,204.807,-58.269,-177.567,6.422,148.451
C06260=1204.315,204.558,-58.245,-177.570,6.420,148.451
C06261=1204.320,204.309,-58.220,-177.573,6.419,148.452
C06262=1204.324,204.060,-58.197,-177.575,6.417,148.452
C06263=1204.329,203.812,-58.173,-177.578,6.415,148.452
C06264=1204.333,203.563,-58.149,-177.581,6.413,148.453
C06265=1204.339,203.314,-58.125,-177.583,6.411,148.453
C06266=1204.343,203.065,-58.101,-177.585,6.409,148.453
C06267=1204.347,202.816,-58.076,-177.588,6.407,148.454
C06268=1204.351,202.567,-58.053,-177.591,6.406,148.454
C06269=1204.356,202.319,-58.029,-177.593,6.404,148.454
C06270=1204.361,202.070,-58.006,-177.596,6.402,148.455
C06271=1204.366,201.821,-57.981,-177.599,6.400,148.455
C06272=1204.370,201.572,-57.958,-177.601,6.398,148.455
C06273=1204.375,201.324,-57.933,-177.604,6.396,148.456
C06274=1204.379,201.075,-57.910,-177.607,6.395,148.456
C06275=1204.384,200.826,-57.886,-177.609,6.393,148.456
C06276=1204.388,200.577,-57.862,-177.612,6.391,148.457
C06277=1204.392,200.328,-57.838,-177.615,6.389,148.457
C06278=1204.397,200.079,-57.815,-177.617,6.387,148.457
C06279=1204.402,199.830,-57.790,-177.620,6.385,148.458
C06280=1204.407,199.581,-57.767,-177.622,6.384,148.458
C06281=1204.411,199.333,-57.743,-177.625,6.382,148.458
C06282=1204.416,199.084,-57.719,-177.627,6.380,148.458
C06283=1204.420,198.835,-57.695,-177.630,6.378,148.459
C06284=1204.425,198.586,-57.672,-177.633,6.376,148.459
C06285=1204.429,198.338,-57.648,-177.635,6.374,148.459
C06286=1204.434,198.089,-57.625,-177.637,6.373,148.460
C06287=1204.439,197.840,-57.601,-177.640,6.371,148.460
C06288=1204.443,197.592,-57.577,-177.643,6.370,148.461
C06289=1204.448,197.343,-57.554,-177.645,6.368,148.461
C06290=1204.453,197.093,-57.530,-177.648,6.366,148.461
C06291=1204.457,196.845,-57.506,-177.651,6.364,148.462
C06292=1204.462,196.596,-57.483,-177.653,6.362,148.462
C06293=1204.466,196.347,-57.460,-177.656,6.360,148.462
C06294=1204.471,196.099,-57.436,-177.659,6.359,148.463
C06295=1204.476,195.850,-57.412,-177.661,6.357,148.463
C06296=1204.480,195.601,-57.389,-177.664,6.355,148.463
C06297=1204.485,195.352,-57.365,-177.667,6.353,148.464
C06298=1204.489,195.103,-57.341,-177.669,6.351,148.464
C06299=1204.494,194.854,-57.318,-177.672,6.350,148.464
C06300=1204.499,194.605,-57.295,-177.674,6.348,148.465
C06301=1204.503,194.357,-57.271,-177.677,6.346,148.465
C06302=1204.508,194.108,-57.247,-177.680,6.344,148.465
C06303=1204.512,193.859,-57.224,-177.682,6.342,148.466
C06304=1204.517,193.609,-57.201,-177.685,6.340,148.466
C06305=1204.521,193.361,-57.178,-177.688,6.339,148.466
C06306=1204.526,193.112,-57.154,-177.690,6.337,148.467
C06307=1204.530,192.863,-57.130,-177.693,6.335,148.467
C06308=1204.535,192.614,-57.107,-177.695,6.334,148.468
C06309=1204.540,192.365,-57.084,-177.698,6.332,148.468
C06310=1204.544,192.116,-57.060,-177.700,6.330,148.468
C06311=1204.549,191.867,-57.037,-177.703,6.329,148.469
C06312=1204.554,191.618,-57.014,-177.706,6.327,148.469
C06313=1204.558,191.369,-56.990,-177.708,6.325,148.469
C06314=1204.562,191.121,-56.967,-177.711,6.323,148.470
C06315=1204.567,190.873,-56.944,-177.714,6.321,148.470
C06316=1204.572,190.624,-56.920,-177.716,6.319,148.470
C06317=1204.577,190.375,-56.897,-177.719,6.318,148.471
C06318=1204.582,190.126,-56.874,-177.722,6.316,148.471
C06319=1204.585,189.877,-56.851,-177.724,6.314,148.471
C06320=1204.590,189.628,-56.827,-177.727,6.312,148.472
C06321=1204.595,189.379,-56.804,-177.729,6.311,148.472
C06322=1204.600,189.130,-56.781,-177.732,6.309,148.472
C06323=1204.604,188.881,-56.757,-177.734,6.308,148.473
C06324=1204.609,188.633,-56.735,-177.737,6.306,148.473
C06325=1204.614,188.384,-56.712,-177.740,6.304,148.474
C06326=1204.618,188.135,-56.688,-177.742,6.302,148.474
C06327=1204.623,187.886,-56.665,-177.745,6.300,148.474
C06328=1204.627,187.637,-56.642,-177.748,6.299,148.475
C06329=1204.632,187.388,-56.619,-177.750,6.297,148.475
C06330=1204.637,187.138,-56.596,-177.753,6.295,148.475
C06331=1204.642,186.890,-56.573,-177.756,6.293,148.476
C06332=1204.646,186.641,-56.550,-177.758,6.292,148.476
C06333=1204.651,186.392,-56.527,-177.760,6.290,148.476
C06334=1204.655,186.143,-56.504,-177.763,6.288,148.477
C06335=1204.659,185.894,-56.481,-177.766,6.287,148.477
C06336=1204.664,185.645,-56.458,-177.768,6.285,148.477
C06337=1204.669,185.376,-56.433,-177.771,6.283,148.478
C06338=1204.674,185.106,-56.408,-177.774,6.282,148.478
C06339=1204.679,184.836,-56.383,-177.777,6.280,148.479
C06340=1204.684,184.567,-56.358,-177.779,6.278,148.479
C06341=1204.689,184.319,-56.336,-177.782,6.276,148.479
C06342=1204.694,184.070,-56.312,-177.785,6.274,148.480
C06343=1204.698,183.820,-56.290,-177.787,6.272,148.480
C06344=1204.703,183.571,-56.267,-177.790,6.271,148.480
C06345=1204.707,183.322,-56.244,-177.793,6.269,148.481
C06346=1204.712,183.074,-56.221,-177.795,6.267,148.481
C06347=1204.717,182.824,-56.198,-177.798,6.265,148.482
C06348=1204.721,182.576,-56.176,-177.800,6.264,148.482
C06349=1204.726,182.327,-56.152,-177.803,6.262,148.482
C06350=1204.731,182.078,-56.130,-177.806,6.261,148.483
C06351=1204.735,181.829,-56.107,-177.809,6.259,148.483
C06352=1204.740,181.580,-56.084,-177.811,6.257,148.484
C06353=1204.744,181.331,-56.061,-177.814,6.256,148.484
C06354=1204.749,181.082,-56.039,-177.817,6.254,148.484
C06355=1204.753,180.834,-56.016,-177.819,6.253,148.485
C06356=1204.758,180.584,-55.994,-177.821,6.251,148.485
C06357=1204.762,180.335,-55.971,-177.824,6.249,148.485
C06358=1204.768,180.087,-55.948,-177.827,6.247,148.486
C06359=1204.772,179.838,-55.926,-177.829,6.245,148.486
C06360=1204.777,179.589,-55.902,-177.832,6.244,148.486
C06361=1204.782,179.340,-55.881,-177.835,6.242,148.487
C06362=1204.786,179.091,-55.857,-177.837,6.241,148.487
C06363=1204.790,178.842,-55.835,-177.839,6.239,148.488
C06364=1204.796,178.593,-55.812,-177.843,6.238,148.488
C06365=1204.800,178.344,-55.789,-177.845,6.236,148.488
C06366=1204.805,178.095,-55.767,-177.848,6.234,148.489
C06367=1204.809,177.846,-55.744,-177.851,6.232,148.489
C06368=1204.814,177.597,-55.722,-177.853,6.231,148.490
C06369=1204.818,177.348,-55.699,-177.855,6.229,148.490
C06370=1204.823,177.099,-55.676,-177.858,6.228,148.490
C06371=1204.828,176.851,-55.654,-177.861,6.226,148.491
C06372=1204.832,176.601,-55.632,-177.863,6.224,148.491
C06373=1204.837,176.353,-55.609,-177.866,6.222,148.491
C06374=1204.842,176.104,-55.587,-177.868,6.221,148.492
C06375=1204.847,175.854,-55.564,-177.871,6.220,148.492
C06376=1204.851,175.606,-55.542,-177.874,6.218,148.493
C06377=1204.856,175.357,-55.520,-177.877,6.216,148.493
C06378=1204.860,175.108,-55.496,-177.879,6.214,148.493
C06379=1204.865,174.859,-55.475,-177.882,6.212,148.494
C06380=1204.870,174.609,-55.452,-177.884,6.211,148.494
C06381=1204.874,174.361,-55.429,-177.887,6.210,148.495
C06382=1204.879,174.112,-55.408,-177.889,6.208,148.495
C06383=1204.884,173.863,-55.384,-177.892,6.206,148.495
C06384=1204.889,173.614,-55.363,-177.895,6.205,148.496
C06385=1204.893,173.365,-55.341,-177.897,6.204,148.496
C06386=1204.898,173.117,-55.318,-177.900,6.202,148.497
C06387=1204.902,172.867,-55.296,-177.903,6.200,148.497
C06388=1204.907,172.618,-55.274,-177.905,6.198,148.497
C06389=1204.912,172.369,-55.251,-177.908,6.196,148.498
C06390=1204.916,172.120,-55.228,-177.910,6.195,148.498
C06391=1204.921,171.872,-55.207,-177.913,6.194,148.498
C06392=1204.925,171.622,-55.185,-177.916,6.192,148.499
C06393=1204.931,171.373,-55.162,-177.918,6.190,148.499
C06394=1204.935,171.125,-55.140,-177.921,6.189,148.500
C06395=1204.939,170.875,-55.118,-177.923,6.188,148.500
C06396=1204.944,170.627,-55.096,-177.926,6.186,148.500
C06397=1204.949,170.377,-55.073,-177.929,6.184,148.501
C06398=1204.954,170.128,-55.052,-177.931,6.182,148.501
C06399=1204.958,169.880,-55.029,-177.934,6.180,148.502
C06400=1204.963,169.631,-55.007,-177.936,6.180,148.502
C06401=1204.968,169.381,-54.985,-177.939,6.178,148.503
C06402=1204.973,169.133,-54.963,-177.942,6.176,148.503
C06403=1204.977,168.883,-54.941,-177.944,6.174,148.503
C06404=1204.982,168.635,-54.919,-177.947,6.173,148.504
C06405=1204.986,168.385,-54.897,-177.949,6.172,148.504
C06406=1204.991,168.137,-54.874,-177.952,6.170,148.505
C06407=1204.996,167.888,-54.852,-177.955,6.168,148.505
C06408=1205.000,167.639,-54.830,-177.958,6.166,148.505
C06409=1205.005,167.390,-54.808,-177.960,6.165,148.506
C06410=1205.010,167.141,-54.787,-177.963,6.164,148.506
C06411=1205.014,166.892,-54.765,-177.965,6.162,148.506
C06412=1205.019,166.643,-54.742,-177.968,6.160,148.507
C06413=1205.024,166.394,-54.720,-177.970,6.159,148.507
C06414=1205.029,166.145,-54.699,-177.973,6.158,148.508
C06415=1205.033,165.896,-54.677,-177.976,6.156,148.508
C06416=1205.038,165.647,-54.655,-177.978,6.154,148.509
C06417=1205.042,165.398,-54.633,-177.981,6.153,148.509
C06418=1205.047,165.149,-54.611,-177.983,6.151,148.509
C06419=1205.052,164.900,-54.589,-177.986,6.150,148.510
C06420=1205.056,164.651,-54.567,-177.989,6.148,148.510
C06421=1205.061,164.402,-54.546,-177.991,6.147,148.511
C06422=1205.065,164.153,-54.524,-177.994,6.145,148.511
C06423=1205.070,163.904,-54.502,-177.996,6.143,148.511
C06424=1205.075,163.655,-54.479,-178.000,6.142,148.512
C06425=1205.080,163.406,-54.458,-178.002,6.141,148.512
C06426=1205.085,163.157,-54.437,-178.004,6.139,148.513
C06427=1205.089,162.907,-54.415,-178.007,6.137,148.513
C06428=1205.094,162.659,-54.393,-178.010,6.136,148.513
C06429=1205.098,162.409,-54.371,-178.012,6.135,148.514
C06430=1205.103,162.161,-54.349,-178.015,6.133,148.514
C06431=1205.108,161.912,-54.328,-178.018,6.131,148.515
C06432=1205.112,161.663,-54.305,-178.020,6.130,148.515
C06433=1205.118,161.414,-54.285,-178.022,6.129,148.516
C06434=1205.122,161.164,-54.262,-178.025,6.127,148.516
C06435=1205.127,160.916,-54.241,-178.028,6.125,148.517
C06436=1205.132,160.667,-54.219,-178.030,6.124,148.517
C06437=1205.136,160.418,-54.197,-178.033,6.123,148.517
C06438=1205.140,160.169,-54.177,-178.036,6.121,148.518
C06439=1205.145,159.920,-54.155,-178.038,6.119,148.518
C06440=1205.150,159.671,-54.133,-178.041,6.118,148.519
C06441=1205.155,159.401,-54.110,-178.044,6.117,148.519
C06442=1205.159,159.133,-54.086,-178.046,6.115,148.519
C06443=1205.165,158.864,-54.063,-178.049,6.113,148.520
C06444=1205.170,158.594,-54.039,-178.052,6.111,148.520
C06445=1205.175,158.346,-54.018,-178.055,6.110,148.521
C06446=1205.180,158.097,-53.997,-178.057,6.109,148.521
C06447=1205.184,157.847,-53.975,-178.060,6.107,148.522
C06448=1205.189,157.599,-53.954,-178.063,6.105,148.522
C06449=1205.194,157.349,-53.933,-178.065,6.104,148.522
C06450=1205.198,157.100,-53.911,-178.068,6.103,148.523
C06451=1205.203,156.851,-53.889,-178.071,6.101,148.523
C06452=1205.208,156.602,-53.868,-178.073,6.099,148.524
C06453=1205.212,156.354,-53.847,-178.075,6.098,148.524
C06454=1205.217,156.104,-53.825,-178.078,6.097,148.525
C06455=1205.222,155.855,-53.804,-178.081,6.095,148.525
C06456=1205.227,155.607,-53.782,-178.083,6.094,148.526
C06457=1205.231,155.357,-53.761,-178.086,6.092,148.526
C06458=1205.236,155.108,-53.739,-178.089,6.091,148.526
C06459=1205.241,154.859,-53.719,-178.091,6.090,148.527
C06460=1205.246,154.610,-53.697,-178.094,6.088,148.527
C06461=1205.250,154.361,-53.675,-178.097,6.086,148.528
C06462=1205.255,154.112,-53.654,-178.099,6.085,148.528
C06463=1205.260,153.863,-53.632,-178.102,6.084,148.529
C06464=1205.264,153.614,-53.612,-178.105,6.082,148.529
C06465=1205.269,153.365,-53.590,-178.107,6.080,148.529
C06466=1205.274,153.116,-53.569,-178.109,6.079,148.530
C06467=1205.279,152.866,-53.548,-178.113,6.078,148.530
C06468=1205.283,152.618,-53.527,-178.115,6.076,148.531
C06469=1205.288,152.368,-53.506,-178.117,6.075,148.531
C06470=1205.292,152.119,-53.484,-178.120,6.073,148.532
C06471=1205.297,151.870,-53.464,-178.123,6.072,148.532
C06472=1205.302,151.622,-53.442,-178.125,6.071,148.533
C06473=1205.307,151.373,-53.421,-178.128,6.069,148.533
C06474=1205.312,151.123,-53.400,-178.131,6.067,148.533
C06475=1205.316,150.874,-53.379,-178.133,6.067,148.534
C06476=1205.321,150.625,-53.358,-178.136,6.065,148.534
C06477=1205.326,150.376,-53.336,-178.138,6.064,148.535
C06478=1205.330,150.127,-53.315,-178.141,6.062,148.535
C06479=1205.335,149.878,-53.295,-178.144,6.061,148.536
C06480=1205.340,149.629,-53.272,-178.146,6.060,148.536
C06481=1205.344,149.380,-53.252,-178.149,6.058,148.536
C06482=1205.349,149.131,-53.231,-178.152,6.057,148.537
C06483=1205.354,148.882,-53.209,-178.154,6.056,148.537
C06484=1205.358,148.633,-53.189,-178.157,6.054,148.538
C06485=1205.364,148.384,-53.168,-178.159,6.052,148.538
C06486=1205.368,148.134,-53.147,-178.162,6.051,148.539
C06487=1205.372,147.885,-53.126,-178.165,6.050,148.539
C06488=1205.378,147.636,-53.105,-178.167,6.048,148.540
C06489=1205.382,147.387,-53.084,-178.169,6.047,148.540
C06490=1205.387,147.138,-53.063,-178.172,6.045,148.541
C06491=1205.391,146.890,-53.042,-178.175,6.044,148.541
C06492=1205.396,146.640,-53.021,-178.177,6.043,148.541
C06493=1205.401,146.390,-53.000,-178.180,6.041,148.542
C06494=1205.405,146.141,-52.980,-178.183,6.040,148.542
C06495=1205.411,145.892,-52.959,-178.185,6.039,148.543
C06496=1205.415,145.644,-52.938,-178.188,6.037,148.543
C06497=1205.420,145.395,-52.917,-178.191,6.036,148.544
C06498=1205.424,145.146,-52.896,-178.193,6.034,148.544
C06499=1205.430,144.896,-52.875,-178.196,6.033,148.545
C06500=1205.434,144.647,-52.855,-178.198,6.032,148.545
C06501=1205.439,144.398,-52.834,-178.201,6.030,148.546
C06502=1205.443,144.150,-52.813,-178.203,6.029,148.546
C06503=1205.448,143.901,-52.792,-178.206,6.028,148.547
C06504=1205.452,143.651,-52.771,-178.209,6.026,148.547
C06505=1205.457,143.402,-52.750,-178.211,6.025,148.547
C06506=1205.462,143.153,-52.730,-178.214,6.024,148.548
C06507=1205.467,142.903,-52.709,-178.216,6.023,148.548
C06508=1205.472,142.655,-52.688,-178.219,6.021,148.549
C06509=1205.477,142.405,-52.667,-178.222,6.019,148.549
C06510=1205.481,142.156,-52.647,-178.224,6.018,148.550
C06511=1205.486,141.907,-52.626,-178.227,6.017,148.550
C06512=1205.491,141.658,-52.606,-178.229,6.016,148.550
C06513=1205.495,141.409,-52.585,-178.232,6.014,148.551
C06514=1205.500,141.160,-52.564,-178.235,6.012,148.551
C06515=1205.505,140.911,-52.544,-178.237,6.011,148.552
C06516=1205.510,140.662,-52.523,-178.240,6.010,148.552
C06517=1205.514,140.413,-52.503,-178.242,6.009,148.553
C06518=1205.520,140.163,-52.482,-178.245,6.007,148.553
C06519=1205.524,139.915,-52.461,-178.248,6.006,148.554
C06520=1205.528,139.666,-52.441,-178.250,6.005,148.554
C06521=1205.534,139.416,-52.420,-178.253,6.003,148.555
C06522=1205.538,139.167,-52.400,-178.256,6.002,148.555
C06523=1205.543,138.918,-52.379,-178.258,6.001,148.556
C06524=1205.548,138.669,-52.358,-178.261,5.999,148.556
C06525=1205.552,138.420,-52.339,-178.264,5.998,148.557
C06526=1205.557,138.171,-52.318,-178.266,5.997,148.557
C06527=1205.562,137.921,-52.297,-178.268,5.996,148.557
C06528=1205.566,137.672,-52.277,-178.272,5.994,148.558
C06529=1205.571,137.423,-52.257,-178.274,5.993,148.558
C06530=1205.576,137.174,-52.236,-178.276,5.991,148.559
C06531=1205.581,136.925,-52.216,-178.280,5.990,148.559
C06532=1205.585,136.676,-52.196,-178.282,5.989,148.560
C06533=1205.590,136.426,-52.175,-178.284,5.987,148.560
C06534=1205.595,136.178,-52.154,-178.287,5.987,148.561
C06535=1205.599,135.929,-52.134,-178.290,5.985,148.561
C06536=1205.605,135.679,-52.114,-178.292,5.984,148.562
C06537=1205.610,135.430,-52.094,-178.295,5.982,148.562
C06538=1205.614,135.181,-52.073,-178.298,5.981,148.563
C06539=1205.619,134.933,-52.053,-178.300,5.980,148.563
C06540=1205.624,134.683,-52.033,-178.303,5.978,148.564
C06541=1205.629,134.434,-52.012,-178.305,5.977,148.564
C06542=1205.633,134.185,-51.992,-178.308,5.976,148.565
C06543=1205.638,133.936,-51.972,-178.310,5.975,148.565
C06544=1205.642,133.686,-51.952,-178.313,5.973,148.565
C06545=1205.648,133.418,-51.929,-178.316,5.972,148.566
C06546=1205.653,133.149,-51.908,-178.318,5.971,148.567
C06547=1205.658,132.881,-51.886,-178.321,5.969,148.567
C06548=1205.664,132.612,-51.864,-178.325,5.968,148.568
C06549=1205.668,132.363,-51.844,-178.327,5.967,148.568
C06550=1205.673,132.113,-51.824,-178.329,5.965,148.569
C06551=1205.677,131.864,-51.804,-178.332,5.965,148.569
C06552=1205.682,131.615,-51.783,-178.335,5.963,148.570
C06553=1205.687,131.366,-51.763,-178.337,5.961,148.570
C06554=1205.692,131.117,-51.743,-178.340,5.960,148.571
C06555=1205.697,130.868,-51.724,-178.343,5.959,148.571
C06556=1205.701,130.619,-51.703,-178.345,5.958,148.572
C06557=1205.706,130.370,-51.683,-178.348,5.956,148.572
C06558=1205.710,130.120,-51.663,-178.350,5.955,148.572
C06559=1205.716,129.871,-51.642,-178.353,5.954,148.573
C06560=1205.721,129.622,-51.623,-178.355,5.953,148.573
C06561=1205.725,129.373,-51.603,-178.359,5.951,148.574
C06562=1205.730,129.124,-51.583,-178.361,5.950,148.574
C06563=1205.735,128.875,-51.563,-178.363,5.949,148.575
C06564=1205.739,128.625,-51.543,-178.366,5.948,148.575
C06565=1205.744,128.376,-51.523,-178.369,5.946,148.576
C06566=1205.749,128.127,-51.503,-178.371,5.946,148.576
C06567=1205.754,127.878,-51.483,-178.374,5.944,148.577
C06568=1205.758,127.629,-51.463,-178.376,5.943,148.577
C06569=1205.763,127.380,-51.443,-178.379,5.942,148.578
C06570=1205.768,127.131,-51.424,-178.381,5.941,148.578
C06571=1205.773,126.881,-51.404,-178.385,5.939,148.579
C06572=1205.777,126.633,-51.384,-178.387,5.938,148.579
C06573=1205.782,126.383,-51.364,-178.389,5.936,148.580
C06574=1205.786,126.134,-51.344,-178.392,5.936,148.580
C06575=1205.792,125.885,-51.324,-178.395,5.934,148.581
C06576=1205.797,125.636,-51.305,-178.397,5.933,148.581
C06577=1205.801,125.387,-51.284,-178.400,5.932,148.582
C06578=1205.806,125.137,-51.265,-178.402,5.931,148.582
C06579=1205.811,124.888,-51.245,-178.405,5.929,148.583
C06580=1205.815,124.639,-51.225,-178.407,5.928,148.583
C06581=1205.820,124.390,-51.205,-178.411,5.927,148.584
C06582=1205.825,124.140,-51.186,-178.413,5.926,148.584
C06583=1205.830,123.892,-51.166,-178.415,5.924,148.585
C06584=1205.835,123.642,-51.146,-178.418,5.924,148.585
C06585=1205.840,123.393,-51.126,-178.421,5.922,148.586
C06586=1205.845,123.144,-51.106,-178.423,5.921,148.586
C06587=1205.849,122.895,-51.087,-178.426,5.919,148.587
C06588=1205.854,122.645,-51.067,-178.429,5.919,148.587
C06589=1205.859,122.396,-51.047,-178.431,5.917,148.588
C06590=1205.864,122.148,-51.027,-178.433,5.916,148.588
C06591=1205.869,121.898,-51.008,-178.437,5.915,148.589
C06592=1205.873,121.648,-50.988,-178.439,5.914,148.589
C06593=1205.878,121.400,-50.969,-178.442,5.912,148.590
C06594=1205.883,121.150,-50.950,-178.444,5.911,148.590
C06595=1205.887,120.901,-50.929,-178.447,5.910,148.591
C06596=1205.892,120.652,-50.910,-178.449,5.909,148.591
C06597=1205.897,120.403,-50.890,-178.452,5.908,148.592
C06598=1205.902,120.153,-50.871,-178.455,5.907,148.592
C06599=1205.907,119.904,-50.851,-178.457,5.906,148.593
C06600=1205.911,119.655,-50.832,-178.460,5.904,148.593
C06601=1205.916,119.406,-50.812,-178.462,5.903,148.594
C06602=1205.921,119.157,-50.793,-178.465,5.902,148.594
C06603=1205.926,118.908,-50.773,-178.467,5.901,148.595
C06604=1205.931,118.658,-50.753,-178.470,5.900,148.595
C06605=1205.936,118.409,-50.734,-178.473,5.899,148.596
C06606=1205.940,118.160,-50.715,-178.476,5.897,148.596
C06607=1205.945,117.911,-50.695,-178.478,5.896,148.597
C06608=1205.950,117.662,-50.676,-178.481,5.894,148.597
C06609=1205.955,117.412,-50.656,-178.483,5.894,148.598
C06610=1205.960,117.163,-50.637,-178.485,5.893,148.598
C06611=1205.964,116.914,-50.618,-178.488,5.891,148.599
C06612=1205.969,116.664,-50.598,-178.491,5.891,148.599
C06613=1205.974,116.416,-50.579,-178.494,5.889,148.600
C06614=1205.979,116.166,-50.559,-178.496,5.888,148.600
C06615=1205.983,115.917,-50.541,-178.499,5.887,148.601
C06616=1205.988,115.668,-50.521,-178.501,5.886,148.601
C06617=1205.993,115.418,-50.501,-178.504,5.884,148.602
C06618=1205.998,115.169,-50.482,-178.507,5.883,148.602
C06619=1206.002,114.920,-50.463,-178.509,5.883,148.603
C06620=1206.008,114.671,-50.444,-178.512,5.881,148.603
C06621=1206.012,114.422,-50.424,-178.514,5.880,148.604
C06622=1206.017,114.173,-50.405,-178.517,5.879,148.604
C06623=1206.022,113.924,-50.386,-178.519,5.878,148.605
C06624=1206.027,113.675,-50.366,-178.522,5.876,148.605
C06625=1206.031,113.425,-50.347,-178.525,5.875,148.606
C06626=1206.036,113.176,-50.328,-178.527,5.875,148.607
C06627=1206.041,112.927,-50.308,-178.530,5.873,148.607
C06628=1206.045,112.678,-50.289,-178.532,5.872,148.608
C06629=1206.051,112.428,-50.271,-178.535,5.871,148.608
C06630=1206.056,112.179,-50.251,-178.538,5.870,148.609
C06631=1206.060,111.930,-50.232,-178.540,5.868,148.609
C06632=1206.065,111.681,-50.213,-178.543,5.868,148.610
C06633=1206.070,111.432,-50.193,-178.545,5.867,148.610
C06634=1206.074,111.182,-50.174,-178.548,5.865,148.611
C06635=1206.080,110.933,-50.156,-178.551,5.864,148.611
C06636=1206.085,110.683,-50.136,-178.554,5.863,148.612
C06637=1206.089,110.435,-50.118,-178.556,5.862,148.612
C06638=1206.094,110.185,-50.098,-178.558,5.861,148.613
C06639=1206.099,109.937,-50.079,-178.561,5.860,148.613
C06640=1206.104,109.687,-50.060,-178.564,5.859,148.614
C06641=1206.108,109.438,-50.042,-178.566,5.857,148.614
C06642=1206.113,109.188,-50.022,-178.569,5.857,148.615
C06643=1206.118,108.940,-50.003,-178.571,5.856,148.615
C06644=1206.123,108.690,-49.984,-178.574,5.854,148.616
C06645=1206.128,108.441,-49.965,-178.577,5.853,148.616
C06646=1206.132,108.192,-49.946,-178.580,5.852,148.617
C06647=1206.138,107.942,-49.927,-178.582,5.851,148.617
C06648=1206.142,107.693,-49.908,-178.584,5.851,148.618
C06649=1206.147,107.425,-49.888,-178.588,5.849,148.619
C06650=1206.153,107.156,-49.868,-178.590,5.847,148.619
C06651=1206.157,106.888,-49.847,-178.593,5.847,148.620
C06652=1206.163,106.619,-49.827,-178.596,5.845,148.620
C06653=1206.168,106.370,-49.807,-178.598,5.844,148.621
C06654=1206.173,106.121,-49.789,-178.601,5.844,148.621
C06655=1206.178,105.872,-49.770,-178.604,5.842,148.622
C06656=1206.182,105.623,-49.751,-178.606,5.841,148.622
C06657=1206.187,105.373,-49.733,-178.609,5.840,148.623
C06658=1206.192,105.124,-49.713,-178.611,5.839,148.623
C06659=1206.197,104.875,-49.695,-178.614,5.838,148.624
C06660=1206.202,104.626,-49.676,-178.617,5.837,148.625
C06661=1206.206,104.377,-49.657,-178.619,5.836,148.625
C06662=1206.212,104.127,-49.638,-178.622,5.835,148.626
C06663=1206.216,103.878,-49.619,-178.624,5.833,148.626
C06664=1206.221,103.628,-49.601,-178.627,5.833,148.627
C06665=1206.226,103.380,-49.582,-178.630,5.831,148.627
C06666=1206.230,103.130,-49.564,-178.632,5.831,148.628
C06667=1206.236,102.881,-49.545,-178.635,5.830,148.628
C06668=1206.240,102.631,-49.526,-178.637,5.828,148.629
C06669=1206.245,102.382,-49.507,-178.640,5.828,148.629
C06670=1206.250,102.133,-49.489,-178.642,5.827,148.630
C06671=1206.254,101.884,-49.470,-178.645,5.825,148.630
C06672=1206.260,101.634,-49.451,-178.648,5.824,148.631
C06673=1206.264,101.386,-49.433,-178.650,5.824,148.632
C06674=1206.269,101.136,-49.414,-178.653,5.822,148.632
C06675=1206.274,100.886,-49.396,-178.655,5.821,148.633
C06676=1206.279,100.638,-49.377,-178.658,5.820,148.633
C06677=1206.283,100.388,-49.359,-178.661,5.819,148.634
C06678=1206.289,100.139,-49.339,-178.663,5.818,148.634
C06679=1206.293,99.890,-49.321,-178.666,5.818,148.635
C06680=1206.298,99.640,-49.303,-178.669,5.816,148.635
C06681=1206.303,99.391,-49.284,-178.671,5.815,148.636
C06682=1206.308,99.142,-49.266,-178.673,5.815,148.636
C06683=1206.312,98.892,-49.247,-178.676,5.813,148.637
C06684=1206.318,98.643,-49.228,-178.679,5.812,148.637
C06685=1206.323,98.394,-49.210,-178.681,5.811,148.638
C06686=1206.327,98.144,-49.192,-178.684,5.810,148.639
C06687=1206.332,97.896,-49.173,-178.686,5.809,148.639
C06688=1206.337,97.646,-49.154,-178.689,5.808,148.640
C06689=1206.342,97.397,-49.137,-178.692,5.807,148.640
C06690=1206.346,97.148,-49.117,-178.694,5.806,148.641
C06691=1206.351,96.899,-49.099,-178.697,5.805,148.641
C06692=1206.357,96.649,-49.081,-178.700,5.804,148.642
C06693=1206.362,96.400,-49.063,-178.702,5.803,148.642
C06694=1206.366,96.151,-49.044,-178.704,5.802,148.643
C06695=1206.370,95.901,-49.026,-178.707,5.801,148.643
C06696=1206.376,95.652,-49.007,-178.710,5.800,148.644
C06697=1206.381,95.403,-48.989,-178.712,5.799,148.644
C06698=1206.385,95.154,-48.970,-178.715,5.798,148.645
C06699=1206.390,94.904,-48.952,-178.718,5.797,148.646
C06700=1206.395,94.655,-48.934,-178.720,5.796,148.646
C06701=1206.401,94.406,-48.916,-178.723,5.795,148.647
C06702=1206.405,94.156,-48.897,-178.725,5.794,148.647
C06703=1206.409,93.907,-48.879,-178.728,5.793,148.648
C06704=1206.414,93.658,-48.861,-178.731,5.792,148.648
C06705=1206.419,93.409,-48.843,-178.733,5.791,148.649
C06706=1206.424,93.159,-48.824,-178.736,5.790,148.649
C06707=1206.429,92.910,-48.806,-178.738,5.790,148.650
C06708=1206.434,92.660,-48.788,-178.741,5.788,148.651
C06709=1206.439,92.411,-48.770,-178.743,5.787,148.651
C06710=1206.444,92.162,-48.752,-178.746,5.787,148.652
C06711=1206.448,91.912,-48.734,-178.749,5.785,148.652
C06712=1206.453,91.664,-48.715,-178.751,5.784,148.653
C06713=1206.458,91.414,-48.697,-178.754,5.783,148.653
C06714=1206.463,91.165,-48.679,-178.757,5.782,148.654
C06715=1206.468,90.916,-48.661,-178.759,5.782,148.655
C06716=1206.473,90.667,-48.642,-178.762,5.781,148.655
C06717=1206.478,90.417,-48.624,-178.764,5.780,148.656
C06718=1206.482,90.168,-48.606,-178.767,5.778,148.656
C06719=1206.487,89.918,-48.588,-178.769,5.778,148.657
C06720=1206.492,89.669,-48.570,-178.772,5.777,148.657
C06721=1206.497,89.420,-48.552,-178.775,5.775,148.658
C06722=1206.502,89.171,-48.534,-178.777,5.775,148.658
C06723=1206.507,88.922,-48.516,-178.780,5.774,148.659
C06724=1206.511,88.672,-48.498,-178.782,5.773,148.659
C06725=1206.516,88.423,-48.480,-178.785,5.772,148.660
C06726=1206.521,88.173,-48.462,-178.787,5.771,148.661
C06727=1206.526,87.924,-48.444,-178.790,5.770,148.661
C06728=1206.531,87.675,-48.426,-178.793,5.769,148.662
C06729=1206.536,87.426,-48.408,-178.795,5.768,148.662
C06730=1206.541,87.176,-48.391,-178.798,5.767,148.663
C06731=1206.546,86.927,-48.373,-178.800,5.767,148.663
C06732=1206.550,86.677,-48.354,-178.803,5.765,148.664
C06733=1206.555,86.428,-48.336,-178.806,5.764,148.664
C06734=1206.560,86.179,-48.318,-178.808,5.764,148.665
C06735=1206.565,85.930,-48.300,-178.811,5.763,148.666
C06736=1206.570,85.680,-48.282,-178.813,5.761,148.666
C06737=1206.575,85.431,-48.264,-178.816,5.761,148.667
C06738=1206.580,85.181,-48.247,-178.819,5.760,148.667
C06739=1206.585,84.932,-48.229,-178.821,5.759,148.668
C06740=1206.590,84.683,-48.211,-178.824,5.758,148.668
C06741=1206.595,84.434,-48.193,-178.826,5.757,148.669
C06742=1206.600,84.185,-48.175,-178.829,5.756,148.670
C06743=1206.604,83.936,-48.158,-178.831,5.756,148.670
C06744=1206.609,83.685,-48.140,-178.834,5.754,148.671
C06745=1206.613,83.436,-48.122,-178.837,5.753,148.671
C06746=1206.618,83.187,-48.104,-178.839,5.753,148.672
C06747=1206.623,82.938,-48.086,-178.842,5.752,148.672
C06748=1206.629,82.688,-48.069,-178.845,5.751,148.673
C06749=1206.633,82.439,-48.051,-178.847,5.750,148.673
C06750=1206.638,82.190,-48.033,-178.849,5.749,148.674
C06751=1206.643,81.940,-48.015,-178.852,5.749,148.675
C06752=1206.648,81.691,-47.998,-178.855,5.747,148.675
C06753=1206.653,81.423,-47.979,-178.857,5.746,148.676
C06754=1206.658,81.154,-47.960,-178.860,5.746,148.676
C06755=1206.664,80.886,-47.941,-178.863,5.744,148.677
C06756=1206.669,80.618,-47.922,-178.866,5.744,148.678
C06757=1206.674,80.368,-47.905,-178.869,5.742,148.678
C06758=1206.679,80.119,-47.887,-178.871,5.741,148.679
C06759=1206.684,79.870,-47.869,-178.874,5.741,148.679
C06760=1206.689,79.620,-47.852,-178.876,5.740,148.680
C06761=1206.693,79.371,-47.834,-178.879,5.739,148.681
C06762=1206.699,79.121,-47.817,-178.882,5.738,148.681
C06763=1206.704,78.872,-47.799,-178.884,5.737,148.682
C06764=1206.708,78.623,-47.781,-178.887,5.736,148.682
C06765=1206.713,78.374,-47.764,-178.889,5.736,148.683
C06766=1206.718,78.124,-47.746,-178.892,5.734,148.683
C06767=1206.723,77.875,-47.729,-178.895,5.734,148.684
C06768=1206.728,77.625,-47.711,-178.897,5.733,148.684
C06769=1206.732,77.377,-47.693,-178.899,5.732,148.685
C06770=1206.737,77.127,-47.676,-178.902,5.732,148.686
C06771=1206.742,76.878,-47.658,-178.905,5.730,148.686
C06772=1206.748,76.628,-47.641,-178.907,5.729,148.687
C06773=1206.752,76.379,-47.624,-178.910,5.729,148.688
C06774=1206.757,76.129,-47.606,-178.912,5.728,148.688
C06775=1206.762,75.880,-47.588,-178.915,5.727,148.689
C06776=1206.767,75.631,-47.572,-178.918,5.726,148.689
C06777=1206.772,75.382,-47.554,-178.920,5.725,148.690
C06778=1206.777,75.132,-47.537,-178.923,5.724,148.690
C06779=1206.782,74.883,-47.519,-178.925,5.724,148.691
C06780=1206.786,74.634,-47.502,-178.927,5.723,148.691
C06781=1206.791,74.384,-47.484,-178.931,5.721,148.692
C06782=1206.797,74.135,-47.467,-178.933,5.721,148.693
C06783=1206.801,73.885,-47.450,-178.935,5.720,148.693
C06784=1206.806,73.636,-47.432,-178.938,5.719,148.694
C06785=1206.811,73.386,-47.415,-178.941,5.719,148.695
C06786=1206.815,73.137,-47.398,-178.943,5.717,148.695
C06787=1206.821,72.888,-47.381,-178.946,5.717,148.696
C06788=1206.826,72.639,-47.364,-178.949,5.716,148.696
C06789=1206.831,72.390,-47.346,-178.951,5.715,148.697
C06790=1206.836,72.140,-47.329,-178.953,5.714,148.697
C06791=1206.840,71.891,-47.311,-178.957,5.713,148.698
C06792=1206.845,71.641,-47.294,-178.959,5.712,148.698
C06793=1206.850,71.392,-47.277,-178.961,5.712,148.699
C06794=1206.855,71.143,-47.260,-178.964,5.711,148.700
C06795=1206.860,70.893,-47.243,-178.967,5.710,148.700
C06796=1206.865,70.644,-47.226,-178.969,5.710,148.701
C06797=1206.870,70.395,-47.208,-178.972,5.708,148.701
C06798=1206.874,70.145,-47.191,-178.975,5.708,148.702
C06799=1206.879,69.895,-47.174,-178.977,5.707,148.703
C06800=1206.885,69.646,-47.157,-178.979,5.706,148.703
C06801=1206.889,69.397,-47.140,-178.982,5.706,148.704
C06802=1206.895,69.148,-47.122,-178.985,5.704,148.704
C06803=1206.899,68.898,-47.106,-178.987,5.703,148.705
C06804=1206.904,68.648,-47.088,-178.990,5.703,148.706
C06805=1206.909,68.399,-47.071,-178.992,5.702,148.706
C06806=1206.914,68.150,-47.054,-178.995,5.701,148.707
C06807=1206.919,67.901,-47.038,-178.997,5.701,148.707
C06808=1206.924,67.651,-47.020,-179.000,5.700,148.708
C06809=1206.928,67.402,-47.003,-179.003,5.698,148.708
C06810=1206.933,67.152,-46.986,-179.005,5.698,148.709
C06811=1206.939,66.904,-46.969,-179.008,5.697,148.710
C06812=1206.944,66.654,-46.952,-179.010,5.696,148.710
C06813=1206.948,66.404,-46.935,-179.013,5.696,148.711
C06814=1206.953,66.155,-46.918,-179.015,5.695,148.712
C06815=1206.958,65.906,-46.901,-179.018,5.694,148.712
C06816=1206.963,65.657,-46.884,-179.021,5.693,148.713
C06817=1206.968,65.407,-46.867,-179.023,5.692,148.713
C06818=1206.972,65.158,-46.850,-179.025,5.692,148.714
C06819=1206.978,64.908,-46.833,-179.028,5.691,148.714
C06820=1206.983,64.659,-46.817,-179.031,5.690,148.715
C06821=1206.988,64.409,-46.800,-179.033,5.690,148.716
C06822=1206.992,64.160,-46.783,-179.036,5.688,148.716
C06823=1206.997,63.911,-46.767,-179.039,5.688,148.717
C06824=1207.003,63.661,-46.749,-179.041,5.687,148.718
C06825=1207.007,63.412,-46.732,-179.044,5.686,148.718
C06826=1207.012,63.163,-46.715,-179.046,5.686,148.719
C06827=1207.017,62.914,-46.698,-179.049,5.685,148.719
C06828=1207.022,62.664,-46.682,-179.051,5.684,148.720
C06829=1207.027,62.415,-46.665,-179.054,5.683,148.720
C06830=1207.031,62.165,-46.648,-179.057,5.682,148.721
C06831=1207.037,61.916,-46.631,-179.059,5.682,148.722
C06832=1207.042,61.666,-46.614,-179.062,5.681,148.722
C06833=1207.046,61.417,-46.598,-179.064,5.680,148.723
C06834=1207.052,61.168,-46.581,-179.067,5.680,148.723
C06835=1207.056,60.918,-46.564,-179.069,5.679,148.724
C06836=1207.061,60.669,-46.547,-179.072,5.678,148.725
C06837=1207.067,60.420,-46.530,-179.075,5.677,148.725
C06838=1207.071,60.170,-46.515,-179.077,5.676,148.726
C06839=1207.076,59.920,-46.498,-179.080,5.675,148.726
C06840=1207.082,59.671,-46.481,-179.082,5.675,148.727
C06841=1207.086,59.422,-46.464,-179.085,5.674,148.728
C06842=1207.091,59.172,-46.448,-179.087,5.674,148.728
C06843=1207.096,58.923,-46.431,-179.090,5.673,148.729
C06844=1207.101,58.674,-46.414,-179.092,5.672,148.729
C06845=1207.106,58.424,-46.397,-179.095,5.671,148.730
C06846=1207.111,58.175,-46.381,-179.098,5.670,148.731
C06847=1207.116,57.926,-46.364,-179.100,5.669,148.731
C06848=1207.121,57.675,-46.348,-179.103,5.669,148.732
C06849=1207.126,57.427,-46.332,-179.106,5.668,148.733
C06850=1207.130,57.177,-46.315,-179.108,5.667,148.733
C06851=1207.136,56.928,-46.298,-179.110,5.667,148.734
C06852=1207.140,56.679,-46.281,-179.113,5.666,148.734
C06853=1207.145,56.429,-46.265,-179.116,5.666,148.735
C06854=1207.150,56.180,-46.249,-179.118,5.665,148.735
C06855=1207.156,55.930,-46.232,-179.121,5.663,148.736
C06856=1207.160,55.680,-46.215,-179.124,5.663,148.737
C06857=1207.165,55.413,-46.197,-179.126,5.662,148.737
C06858=1207.171,55.144,-46.180,-179.129,5.662,148.738
C06859=1207.176,54.875,-46.162,-179.131,5.661,148.739
C06860=1207.182,54.607,-46.145,-179.135,5.660,148.739
C06861=1207.186,54.357,-46.128,-179.137,5.659,148.740
C06862=1207.191,54.108,-46.112,-179.139,5.658,148.740
C06863=1207.196,53.858,-46.096,-179.142,5.658,148.741
C06864=1207.202,53.609,-46.079,-179.145,5.657,148.742
C06865=1207.206,53.360,-46.062,-179.147,5.656,148.742
C06866=1207.211,53.110,-46.045,-179.149,5.656,148.743
C06867=1207.216,52.861,-46.030,-179.152,5.655,148.744
C06868=1207.221,52.611,-46.013,-179.155,5.655,148.744
C06869=1207.226,52.363,-45.997,-179.157,5.654,148.745
C06870=1207.231,52.113,-45.981,-179.160,5.653,148.745
C06871=1207.236,51.864,-45.965,-179.163,5.652,148.746
C06872=1207.241,51.614,-45.947,-179.165,5.651,148.747
C06873=1207.246,51.365,-45.932,-179.168,5.651,148.747
C06874=1207.251,51.115,-45.915,-179.170,5.650,148.748
C06875=1207.256,50.866,-45.900,-179.173,5.649,148.748
C06876=1207.261,50.616,-45.883,-179.175,5.649,148.749
C06877=1207.265,50.367,-45.866,-179.178,5.648,148.750
C06878=1207.271,50.117,-45.851,-179.180,5.647,148.750
C06879=1207.275,49.868,-45.834,-179.183,5.647,148.751
C06880=1207.280,49.618,-45.818,-179.186,5.646,148.752
C06881=1207.285,49.369,-45.802,-179.188,5.646,148.752
C06882=1207.290,49.120,-45.785,-179.190,5.645,148.753
C06883=1207.295,48.870,-45.769,-179.193,5.644,148.753
C06884=1207.300,48.621,-45.753,-179.196,5.643,148.754
C06885=1207.305,48.371,-45.737,-179.199,5.642,148.755
C06886=1207.310,48.122,-45.721,-179.201,5.642,148.755
C06887=1207.315,47.872,-45.705,-179.204,5.641,148.756
C06888=1207.320,47.623,-45.689,-179.206,5.640,148.756
C06889=1207.324,47.373,-45.673,-179.209,5.640,148.757
C06890=1207.329,47.125,-45.656,-179.211,5.639,148.758
C06891=1207.335,46.875,-45.641,-179.214,5.638,148.758
C06892=1207.339,46.626,-45.624,-179.216,5.638,148.759
C06893=1207.345,46.376,-45.609,-179.219,5.637,148.760
C06894=1207.349,46.127,-45.592,-179.221,5.637,148.760
C06895=1207.355,45.877,-45.576,-179.224,5.636,148.761
C06896=1207.359,45.627,-45.560,-179.226,5.635,148.761
C06897=1207.364,45.379,-45.544,-179.229,5.635,148.762
C06898=1207.369,45.128,-45.528,-179.232,5.634,148.763
C06899=1207.374,44.880,-45.512,-179.234,5.633,148.763
C06900=1207.379,44.630,-45.496,-179.236,5.633,148.764
C06901=1207.384,44.381,-45.480,-179.239,5.632,148.765
C06902=1207.390,44.131,-45.464,-179.242,5.632,148.765
C06903=1207.394,43.881,-45.448,-179.244,5.631,148.766
C06904=1207.399,43.632,-45.432,-179.246,5.630,148.766
C06905=1207.404,43.382,-45.416,-179.250,5.629,148.767
C06906=1207.410,43.133,-45.400,-179.252,5.629,148.768
C06907=1207.415,42.884,-45.384,-179.255,5.628,148.768
C06908=1207.419,42.634,-45.368,-179.257,5.627,148.769
C06909=1207.424,42.385,-45.353,-179.260,5.627,148.769
C06910=1207.429,42.135,-45.336,-179.262,5.626,148.770
C06911=1207.434,41.886,-45.321,-179.265,5.625,148.771
C06912=1207.439,41.637,-45.305,-179.268,5.625,148.771
C06913=1207.444,41.387,-45.288,-179.270,5.624,148.772
C06914=1207.449,41.138,-45.273,-179.272,5.623,148.773
C06915=1207.455,40.888,-45.257,-179.275,5.623,148.773
C06916=1207.459,40.638,-45.241,-179.278,5.622,148.774
C06917=1207.464,40.390,-45.226,-179.280,5.622,148.774
C06918=1207.469,40.140,-45.210,-179.283,5.621,148.775
C06919=1207.474,39.890,-45.194,-179.285,5.620,148.776
C06920=1207.479,39.641,-45.178,-179.288,5.620,148.776
C06921=1207.484,39.391,-45.162,-179.290,5.619,148.777
C06922=1207.489,39.142,-45.146,-179.293,5.618,148.778
C06923=1207.494,38.893,-45.131,-179.295,5.618,148.778
C06924=1207.499,38.643,-45.115,-179.298,5.617,148.779
C06925=1207.504,38.393,-45.100,-179.301,5.617,148.780
C06926=1207.509,38.145,-45.083,-179.303,5.616,148.780
C06927=1207.514,37.895,-45.067,-179.305,5.615,148.781
C06928=1207.519,37.645,-45.052,-179.308,5.615,148.781
C06929=1207.524,37.396,-45.037,-179.311,5.614,148.782
C06930=1207.529,37.146,-45.021,-179.313,5.614,148.783
C06931=1207.534,36.897,-45.005,-179.316,5.613,148.783
C06932=1207.538,36.648,-44.990,-179.318,5.612,148.784
C06933=1207.544,36.399,-44.974,-179.321,5.612,148.784
C06934=1207.549,36.149,-44.958,-179.323,5.611,148.785
C06935=1207.554,35.899,-44.942,-179.326,5.611,148.786
C06936=1207.559,35.650,-44.927,-179.329,5.610,148.786
C06937=1207.563,35.400,-44.911,-179.331,5.609,148.787
C06938=1207.569,35.151,-44.896,-179.333,5.609,148.788
C06939=1207.574,34.901,-44.880,-179.336,5.608,148.788
C06940=1207.579,34.652,-44.865,-179.339,5.608,148.789
C06941=1207.584,34.402,-44.849,-179.341,5.607,148.790
C06942=1207.589,34.153,-44.834,-179.344,5.606,148.790
C06943=1207.594,33.903,-44.819,-179.346,5.606,148.791
C06944=1207.598,33.653,-44.803,-179.349,5.605,148.791
C06945=1207.604,33.404,-44.787,-179.351,5.605,148.792
C06946=1207.608,33.155,-44.771,-179.354,5.604,148.793
C06947=1207.614,32.906,-44.756,-179.356,5.603,148.793
C06948=1207.618,32.656,-44.740,-179.359,5.603,148.794
C06949=1207.623,32.407,-44.725,-179.362,5.602,148.795
C06950=1207.629,32.157,-44.710,-179.364,5.602,148.795
C06951=1207.634,31.907,-44.694,-179.367,5.601,148.796
C06952=1207.638,31.658,-44.679,-179.369,5.601,148.797
C06953=1207.644,31.408,-44.664,-179.372,5.600,148.797
C06954=1207.649,31.159,-44.648,-179.374,5.599,148.798
C06955=1207.654,30.910,-44.633,-179.377,5.599,148.798
C06956=1207.659,30.660,-44.617,-179.380,5.598,148.799
C06957=1207.663,30.411,-44.602,-179.382,5.598,148.800
C06958=1207.668,30.161,-44.586,-179.384,5.597,148.800
C06959=1207.674,29.912,-44.571,-179.387,5.596,148.801
C06960=1207.678,29.663,-44.556,-179.390,5.596,148.802
C06961=1207.684,29.394,-44.540,-179.392,5.595,148.802
C06962=1207.689,29.125,-44.523,-179.395,5.595,148.803
C06963=1207.695,28.856,-44.507,-179.398,5.594,148.804
C06964=1207.700,28.587,-44.489,-179.400,5.594,148.804
C06965=1207.705,28.338,-44.474,-179.403,5.593,148.805
C06966=1207.710,28.089,-44.459,-179.405,5.593,148.806
C06967=1207.715,27.840,-44.444,-179.408,5.592,148.806
C06968=1207.720,27.590,-44.429,-179.411,5.592,148.807
C06969=1207.725,27.340,-44.414,-179.413,5.591,148.807
C06970=1207.730,27.090,-44.398,-179.416,5.590,148.808
C06971=1207.735,26.841,-44.382,-179.418,5.590,148.809
C06972=1207.740,26.592,-44.367,-179.421,5.589,148.809
C06973=1207.745,26.342,-44.353,-179.424,5.589,148.810
C06974=1207.750,26.093,-44.338,-179.426,5.588,148.811
C06975=1207.755,25.843,-44.322,-179.428,5.588,148.811
C06976=1207.760,25.594,-44.307,-179.430,5.587,148.812
C06977=1207.765,25.343,-44.292,-179.433,5.587,148.813
C06978=1207.770,25.094,-44.277,-179.436,5.586,148.813
C06979=1207.775,24.845,-44.261,-179.438,5.586,148.814
C06980=1207.780,24.596,-44.246,-179.440,5.585,148.814
C06981=1207.785,24.346,-44.232,-179.443,5.584,148.815
C06982=1207.790,24.097,-44.216,-179.446,5.584,148.816
C06983=1207.795,23.848,-44.201,-179.448,5.583,148.817
C06984=1207.801,23.598,-44.186,-179.451,5.583,148.817
C06985=1207.805,23.348,-44.171,-179.454,5.582,148.818
C06986=1207.810,23.098,-44.156,-179.456,5.582,148.818
C06987=1207.815,22.849,-44.141,-179.459,5.581,148.819
C06988=1207.820,22.599,-44.126,-179.461,5.580,148.820
C06989=1207.825,22.350,-44.111,-179.464,5.580,148.820
C06990=1207.830,22.101,-44.096,-179.466,5.579,148.821
C06991=1207.835,21.851,-44.081,-179.469,5.580,148.822
C06992=1207.840,21.602,-44.066,-179.471,5.579,148.822
C06993=1207.846,21.352,-44.051,-179.473,5.578,148.823
C06994=1207.850,21.103,-44.036,-179.476,5.578,148.824
C06995=1207.855,20.854,-44.021,-179.479,5.577,148.824
C06996=1207.861,20.604,-44.006,-179.481,5.577,148.825
C06997=1207.865,20.355,-43.991,-179.484,5.576,148.826
C06998=1207.871,20.105,-43.976,-179.487,5.576,148.826
C06999=1207.875,19.855,-43.961,-179.489,5.575,148.827
C07000=1207.880,19.606,-43.946,-179.491,5.574,148.827
C07001=1207.885,19.356,-43.931,-179.494,5.574,148.828
C07002=1207.890,19.107,-43.916,-179.497,5.573,148.829
C07003=1207.895,18.857,-43.902,-179.499,5.573,148.829
C07004=1207.900,18.608,-43.886,-179.501,5.573,148.830
C07005=1207.905,18.358,-43.872,-179.504,5.572,148.831
C07006=1207.910,18.109,-43.857,-179.506,5.572,148.831
C07007=1207.916,17.859,-43.842,-179.509,5.571,148.832
C07008=1207.920,17.610,-43.827,-179.511,5.571,148.833
C07009=1207.925,17.360,-43.813,-179.514,5.570,148.833
C07010=1207.930,17.111,-43.798,-179.517,5.570,148.834
C07011=1207.936,16.861,-43.783,-179.519,5.569,148.835
C07012=1207.940,16.612,-43.768,-179.522,5.568,148.835
C07013=1207.945,16.362,-43.754,-179.524,5.568,148.836
C07014=1207.951,16.113,-43.738,-179.527,5.567,148.836
C07015=1207.956,15.863,-43.724,-179.529,5.567,148.837
C07016=1207.961,15.613,-43.709,-179.532,5.567,148.838
C07017=1207.965,15.364,-43.694,-179.534,5.566,148.839
C07018=1207.971,15.114,-43.680,-179.536,5.566,148.839
C07019=1207.976,14.865,-43.665,-179.539,5.565,148.840
C07020=1207.981,14.615,-43.650,-179.542,5.565,148.840
C07021=1207.985,14.366,-43.636,-179.544,5.564,148.841
C07022=1207.991,14.116,-43.620,-179.547,5.564,148.842
C07023=1207.996,13.867,-43.606,-179.550,5.563,148.842
C07024=1208.000,13.617,-43.591,-179.552,5.562,148.843
C07025=1208.005,13.368,-43.577,-179.554,5.562,148.844
C07026=1208.011,13.119,-43.563,-179.557,5.562,148.844
C07027=1208.016,12.869,-43.547,-179.559,5.561,148.845
C07028=1208.021,12.620,-43.533,-179.562,5.561,148.846
C07029=1208.026,12.370,-43.519,-179.564,5.560,148.846
C07030=1208.031,12.121,-43.504,-179.567,5.560,148.847
C07031=1208.036,11.871,-43.490,-179.570,5.559,148.848
C07032=1208.042,11.621,-43.475,-179.572,5.558,148.848
C07033=1208.046,11.372,-43.460,-179.575,5.558,148.849
C07034=1208.051,11.122,-43.445,-179.577,5.558,148.849
C07035=1208.056,10.873,-43.431,-179.579,5.558,148.850
C07036=1208.061,10.623,-43.417,-179.582,5.557,148.851
C07037=1208.066,10.374,-43.402,-179.585,5.557,148.852
C07038=1208.071,10.124,-43.387,-179.587,5.556,148.852
C07039=1208.077,9.875,-43.373,-179.590,5.556,148.853
C07040=1208.082,9.625,-43.359,-179.592,5.555,148.853
C07041=1208.087,9.376,-43.344,-179.595,5.554,148.854
C07042=1208.092,9.126,-43.330,-179.597,5.555,148.855
C07043=1208.096,8.877,-43.315,-179.599,5.554,148.855
C07044=1208.101,8.627,-43.301,-179.602,5.554,148.856
C07045=1208.106,8.377,-43.287,-179.605,5.553,148.857
C07046=1208.111,8.128,-43.272,-179.607,5.553,148.857
C07047=1208.117,7.878,-43.257,-179.610,5.552,148.858
C07048=1208.122,7.629,-43.243,-179.612,5.551,148.859
C07049=1208.127,7.379,-43.229,-179.614,5.551,148.859
C07050=1208.132,7.130,-43.214,-179.617,5.551,148.860
C07051=1208.137,6.880,-43.199,-179.620,5.550,148.861
C07052=1208.142,6.631,-43.185,-179.622,5.550,148.861
C07053=1208.147,6.381,-43.171,-179.625,5.549,148.862
C07054=1208.152,6.131,-43.157,-179.627,5.549,148.863
C07055=1208.157,5.882,-43.143,-179.630,5.548,148.863
C07056=1208.162,5.633,-43.128,-179.632,5.548,148.864
C07057=1208.167,5.383,-43.114,-179.634,5.548,148.865
C07058=1208.172,5.133,-43.100,-179.637,5.547,148.865
C07059=1208.177,4.883,-43.086,-179.640,5.547,148.866
C07060=1208.182,4.634,-43.071,-179.642,5.546,148.867
C07061=1208.187,4.385,-43.057,-179.645,5.546,148.867
C07062=1208.192,4.136,-43.042,-179.647,5.545,148.868
C07063=1208.197,3.886,-43.028,-179.649,5.545,148.868
C07064=1208.202,3.636,-43.014,-179.652,5.545,148.869
C07065=1208.208,3.367,-42.999,-179.655,5.544,148.870
C07066=1208.213,3.099,-42.983,-179.657,5.544,148.871
C07067=1208.219,2.829,-42.969,-179.660,5.543,148.871
C07068=1208.224,2.561,-42.953,-179.663,5.543,148.872
C07069=1208.229,2.311,-42.939,-179.665,5.542,148.873
C07070=1208.234,2.061,-42.924,-179.668,5.542,148.873
C07071=1208.239,1.812,-42.910,-179.670,5.541,148.874
C07072=1208.244,1.562,-42.896,-179.673,5.541,148.875
C07073=1208.249,1.313,-42.882,-179.675,5.541,148.875
C07074=1208.254,1.063,-42.867,-179.678,5.541,148.876
C07075=1208.259,0.813,-42.853,-179.681,5.540,148.877
C07076=1208.265,0.564,-42.840,-179.683,5.540,148.877
C07077=1208.270,0.314,-42.826,-179.685,5.539,148.878
C07078=1208.275,0.064,-42.811,-179.688,5.538,148.879
C07079=1208.280,-0.186,-42.797,-179.691,5.538,148.879
C07080=1208.285,-0.435,-42.783,-179.693,5.538,148.880
C07081=1208.290,-0.684,-42.769,-179.695,5.537,148.881
C07082=1208.295,-0.934,-42.755,-179.698,5.537,148.881
C07083=1208.300,-1.183,-42.741,-179.701,5.536,148.882
C07084=1208.305,-1.432,-42.727,-179.703,5.536,148.883
C07085=1208.310,-1.682,-42.713,-179.705,5.536,148.883
C07086=1208.315,-1.932,-42.699,-179.708,5.535,148.884
C07087=1208.321,-2.181,-42.685,-179.710,5.535,148.885
C07088=1208.326,-2.431,-42.671,-179.713,5.534,148.885
C07089=1208.331,-2.681,-42.657,-179.716,5.534,148.886
C07090=1208.335,-2.930,-42.643,-179.718,5.533,148.887
C07091=1208.341,-3.179,-42.629,-179.720,5.534,148.887
C07092=1208.346,-3.429,-42.615,-179.723,5.533,148.888
C07093=1208.351,-3.679,-42.601,-179.726,5.533,148.889
C07094=1208.356,-3.928,-42.587,-179.728,5.532,148.889
C07095=1208.361,-4.178,-42.573,-179.730,5.531,148.890
C07096=1208.366,-4.427,-42.560,-179.732,5.532,148.891
C07097=1208.371,-4.676,-42.546,-179.735,5.531,148.891
C07098=1208.376,-4.927,-42.532,-179.738,5.531,148.892
C07099=1208.381,-5.176,-42.518,-179.740,5.530,148.893
C07100=1208.387,-5.425,-42.504,-179.743,5.530,148.893
C07101=1208.391,-5.675,-42.490,-179.746,5.529,148.894
C07102=1208.396,-5.925,-42.477,-179.748,5.530,148.895
C07103=1208.402,-6.174,-42.463,-179.750,5.529,148.895
C07104=1208.407,-6.424,-42.448,-179.753,5.528,148.896
C07105=1208.411,-6.673,-42.435,-179.755,5.528,148.897
C07106=1208.417,-6.923,-42.422,-179.758,5.527,148.897
C07107=1208.422,-7.173,-42.407,-179.760,5.527,148.898
C07108=1208.427,-7.422,-42.393,-179.763,5.527,148.899
C07109=1208.432,-7.672,-42.380,-179.765,5.526,148.899
C07110=1208.437,-7.921,-42.366,-179.768,5.526,148.900
C07111=1208.442,-8.171,-42.352,-179.771,5.526,148.901
C07112=1208.448,-8.421,-42.339,-179.772,5.525,148.901
C07113=1208.452,-8.670,-42.325,-179.775,5.525,148.902
C07114=1208.457,-8.920,-42.311,-179.778,5.524,148.902
C07115=1208.463,-9.169,-42.297,-179.780,5.524,148.903
C07116=1208.467,-9.419,-42.284,-179.783,5.523,148.904
C07117=1208.473,-9.668,-42.270,-179.785,5.524,148.905
C07118=1208.478,-9.918,-42.256,-179.788,5.523,148.905
C07119=1208.482,-10.168,-42.243,-179.790,5.523,148.906
C07120=1208.488,-10.417,-42.229,-179.793,5.522,148.907
C07121=1208.493,-10.667,-42.215,-179.795,5.521,148.907
C07122=1208.498,-10.916,-42.202,-179.797,5.522,148.908
C07123=1208.503,-11.166,-42.188,-179.800,5.521,148.908
C07124=1208.508,-11.416,-42.174,-179.802,5.521,148.909
C07125=1208.513,-11.665,-42.161,-179.805,5.520,148.910
C07126=1208.518,-11.915,-42.147,-179.807,5.521,148.911
C07127=1208.524,-12.164,-42.134,-179.810,5.520,148.911
C07128=1208.528,-12.414,-42.120,-179.813,5.520,148.912
C07129=1208.534,-12.663,-42.106,-179.815,5.519,148.913
C07130=1208.538,-12.913,-42.093,-179.817,5.518,148.913
C07131=1208.543,-13.162,-42.079,-179.819,5.519,148.914
C07132=1208.549,-13.412,-42.066,-179.822,5.518,148.914
C07133=1208.553,-13.661,-42.052,-179.825,5.518,148.915
C07134=1208.559,-13.911,-42.039,-179.827,5.517,148.916
C07135=1208.564,-14.161,-42.025,-179.829,5.517,148.917
C07136=1208.569,-14.410,-42.012,-179.832,5.517,148.917
C07137=1208.574,-14.660,-41.998,-179.835,5.516,148.918
C07138=1208.579,-14.909,-41.985,-179.837,5.516,148.919
C07139=1208.584,-15.159,-41.972,-179.840,5.515,148.919
C07140=1208.589,-15.408,-41.958,-179.842,5.515,148.920
C07141=1208.594,-15.659,-41.945,-179.844,5.515,148.921
C07142=1208.600,-15.908,-41.931,-179.847,5.514,148.921
C07143=1208.605,-16.158,-41.918,-179.850,5.514,148.922
C07144=1208.610,-16.407,-41.904,-179.852,5.514,148.923
C07145=1208.615,-16.657,-41.891,-179.854,5.514,148.923
C07146=1208.620,-16.907,-41.878,-179.857,5.513,148.924
C07147=1208.625,-17.156,-41.864,-179.860,5.513,148.925
C07148=1208.630,-17.406,-41.851,-179.862,5.513,148.925
C07149=1208.635,-17.655,-41.837,-179.864,5.512,148.926
C07150=1208.641,-17.904,-41.824,-179.867,5.512,148.927
C07151=1208.645,-18.154,-41.811,-179.869,5.511,148.927
C07152=1208.651,-18.403,-41.797,-179.871,5.512,148.928
C07153=1208.655,-18.653,-41.784,-179.874,5.511,148.929
C07154=1208.661,-18.903,-41.771,-179.877,5.511,148.929
C07155=1208.665,-19.152,-41.757,-179.879,5.510,148.930
C07156=1208.671,-19.402,-41.744,-179.881,5.510,148.931
C07157=1208.676,-19.652,-41.731,-179.884,5.510,148.931
C07158=1208.681,-19.901,-41.717,-179.886,5.509,148.932
C07159=1208.686,-20.151,-41.704,-179.889,5.509,148.933
C07160=1208.692,-20.401,-41.691,-179.891,5.509,148.933
C07161=1208.696,-20.651,-41.678,-179.894,5.508,148.934
C07162=1208.702,-20.900,-41.664,-179.896,5.508,148.935
C07163=1208.707,-21.149,-41.652,-179.899,5.508,148.935
C07164=1208.711,-21.399,-41.639,-179.901,5.508,148.936
C07165=1208.717,-21.648,-41.625,-179.904,5.507,148.937
C07166=1208.721,-21.898,-41.612,-179.906,5.507,148.937
C07167=1208.727,-22.148,-41.599,-179.909,5.506,148.938
C07168=1208.732,-22.398,-41.586,-179.911,5.506,148.939
C07169=1208.738,-22.666,-41.571,-179.914,5.506,148.940
C07170=1208.743,-22.936,-41.557,-179.916,5.506,148.940
C07171=1208.749,-23.206,-41.543,-179.919,5.505,148.941
C07172=1208.755,-23.475,-41.528,-179.922,5.505,148.942
C07173=1208.759,-23.725,-41.516,-179.924,5.504,148.942
C07174=1208.764,-23.974,-41.503,-179.926,5.505,148.943
C07175=1208.770,-24.225,-41.489,-179.929,5.504,148.944
C07176=1208.775,-24.474,-41.477,-179.932,5.504,148.944
C07177=1208.780,-24.723,-41.463,-179.934,5.503,148.945
C07178=1208.785,-24.973,-41.450,-179.936,5.503,148.946
C07179=1208.790,-25.222,-41.437,-179.939,5.503,148.946
C07180=1208.794,-25.472,-41.424,-179.941,5.502,148.947
C07181=1208.800,-25.722,-41.411,-179.944,5.502,148.948
C07182=1208.805,-25.971,-41.399,-179.946,5.502,148.948
C07183=1208.810,-26.221,-41.386,-179.949,5.502,148.949
C07184=1208.815,-26.470,-41.372,-179.951,5.501,148.950
C07185=1208.820,-26.720,-41.359,-179.953,5.501,148.950
C07186=1208.825,-26.970,-41.346,-179.956,5.501,148.951
C07187=1208.831,-27.219,-41.333,-179.958,5.500,148.952
C07188=1208.836,-27.469,-41.320,-179.961,5.500,148.952
C07189=1208.841,-27.718,-41.307,-179.963,5.500,148.953
C07190=1208.846,-27.968,-41.294,-179.966,5.499,148.954
C07191=1208.851,-28.218,-41.281,-179.968,5.499,148.954
C07192=1208.856,-28.467,-41.269,-179.971,5.498,148.955
C07193=1208.861,-28.717,-41.256,-179.973,5.499,148.956
C07194=1208.867,-28.967,-41.242,-179.976,5.498,148.956
C07195=1208.872,-29.216,-41.230,-179.978,5.498,148.957
C07196=1208.877,-29.466,-41.217,-179.980,5.498,148.958
C07197=1208.882,-29.716,-41.204,-179.983,5.497,148.958
C07198=1208.887,-29.965,-41.191,-179.985,5.497,148.959
C07199=1208.892,-30.215,-41.178,-179.988,5.496,148.960
C07200=1208.897,-30.465,-41.165,-179.990,5.497,148.960
C07201=1208.902,-30.714,-41.153,-179.993,5.496,148.961
C07202=1208.908,-30.964,-41.140,-179.995,5.496,148.962
C07203=1208.913,-31.213,-41.127,-179.997,5.496,148.963
C07204=1208.917,-31.463,-41.114,180.000,5.496,148.963
C07205=1208.923,-31.712,-41.101,179.997,5.495,148.964
C07206=1208.928,-31.962,-41.088,179.995,5.495,148.965
C07207=1208.933,-32.212,-41.075,179.993,5.495,148.965
C07208=1208.938,-32.461,-41.063,179.990,5.494,148.966
C07209=1208.943,-32.711,-41.050,179.988,5.494,148.966
C07210=1208.948,-32.960,-41.038,179.986,5.494,148.967
C07211=1208.954,-33.210,-41.024,179.983,5.494,148.968
C07212=1208.959,-33.460,-41.011,179.980,5.493,148.969
C07213=1208.964,-33.710,-40.999,179.978,5.493,148.969
C07214=1208.969,-33.960,-40.987,179.975,5.493,148.970
C07215=1208.974,-34.209,-40.974,179.973,5.492,148.971
C07216=1208.979,-34.458,-40.961,179.970,5.492,148.971
C07217=1208.985,-34.708,-40.948,179.969,5.492,148.972
C07218=1208.989,-34.958,-40.935,179.966,5.491,148.973
C07219=1208.994,-35.207,-40.923,179.963,5.491,148.973
C07220=1209.000,-35.457,-40.911,179.961,5.491,148.974
C07221=1209.005,-35.706,-40.898,179.958,5.491,148.975
C07222=1209.010,-35.956,-40.885,179.956,5.490,148.975
C07223=1209.015,-36.206,-40.872,179.954,5.491,148.976
C07224=1209.020,-36.455,-40.860,179.951,5.490,148.977
C07225=1209.026,-36.705,-40.847,179.948,5.490,148.977
C07226=1209.031,-36.955,-40.835,179.947,5.490,148.978
C07227=1209.036,-37.205,-40.822,179.944,5.489,148.979
C07228=1209.041,-37.454,-40.809,179.942,5.489,148.979
C07229=1209.046,-37.703,-40.797,179.939,5.488,148.980
C07230=1209.051,-37.953,-40.785,179.937,5.489,148.981
C07231=1209.056,-38.203,-40.772,179.934,5.488,148.981
C07232=1209.061,-38.453,-40.759,179.931,5.488,148.982
C07233=1209.066,-38.702,-40.747,179.929,5.488,148.983
C07234=1209.071,-38.952,-40.735,179.927,5.488,148.983
C07235=1209.077,-39.201,-40.722,179.924,5.487,148.984
C07236=1209.082,-39.450,-40.710,179.922,5.487,148.985
C07237=1209.088,-39.700,-40.696,179.920,5.487,148.985
C07238=1209.092,-39.951,-40.684,179.917,5.486,148.986
C07239=1209.097,-40.200,-40.671,179.915,5.486,148.987
C07240=1209.103,-40.449,-40.659,179.912,5.486,148.987
C07241=1209.108,-40.699,-40.647,179.910,5.486,148.988
C07242=1209.113,-40.949,-40.634,179.908,5.486,148.989
C07243=1209.118,-41.198,-40.622,179.905,5.485,148.990
C07244=1209.123,-41.449,-40.610,179.902,5.485,148.990
C07245=1209.128,-41.698,-40.597,179.900,5.485,148.991
C07246=1209.133,-41.947,-40.584,179.898,5.484,148.991
C07247=1209.139,-42.197,-40.572,179.895,5.484,148.992
C07248=1209.144,-42.446,-40.560,179.893,5.484,148.993
C07249=1209.149,-42.696,-40.547,179.891,5.484,148.994
C07250=1209.154,-42.946,-40.535,179.888,5.483,148.994
C07251=1209.159,-43.196,-40.522,179.886,5.484,148.995
C07252=1209.164,-43.445,-40.511,179.883,5.483,148.996
C07253=1209.169,-43.695,-40.498,179.881,5.483,148.996
C07254=1209.174,-43.944,-40.486,179.878,5.483,148.997
C07255=1209.179,-44.194,-40.474,179.876,5.483,148.998
C07256=1209.184,-44.443,-40.461,179.874,5.482,148.998
C07257=1209.190,-44.693,-40.450,179.872,5.482,148.999
C07258=1209.195,-44.942,-40.437,179.869,5.482,149.000
C07259=1209.200,-45.192,-40.425,179.866,5.481,149.000
C07260=1209.205,-45.442,-40.412,179.864,5.482,149.001
C07261=1209.210,-45.692,-40.400,179.861,5.481,149.002
C07262=1209.216,-45.942,-40.388,179.859,5.481,149.002
C07263=1209.221,-46.192,-40.376,179.857,5.481,149.003
C07264=1209.226,-46.441,-40.363,179.854,5.481,149.004
C07265=1209.232,-46.691,-40.351,179.852,5.480,149.004
C07266=1209.236,-46.940,-40.339,179.850,5.480,149.005
C07267=1209.241,-47.190,-40.327,179.847,5.480,149.006
C07268=1209.246,-47.439,-40.315,179.844,5.479,149.006
C07269=1209.252,-47.689,-40.303,179.842,5.479,149.007
C07270=1209.257,-47.938,-40.290,179.840,5.479,149.008
C07271=1209.262,-48.188,-40.278,179.837,5.479,149.009
C07272=1209.268,-48.438,-40.266,179.835,5.479,149.009
C07273=1209.273,-48.708,-40.253,179.832,5.478,149.010
C07274=1209.278,-48.978,-40.240,179.830,5.478,149.011
C07275=1209.284,-49.247,-40.226,179.827,5.477,149.011
C07276=1209.289,-49.518,-40.214,179.825,5.478,149.012
C07277=1209.295,-49.768,-40.202,179.822,5.477,149.013
C07278=1209.300,-50.017,-40.189,179.820,5.477,149.013
C07279=1209.305,-50.267,-40.177,179.817,5.477,149.014
C07280=1209.311,-50.517,-40.165,179.815,5.477,149.015
C07281=1209.315,-50.766,-40.153,179.812,5.476,149.016
C07282=1209.320,-51.016,-40.141,179.810,5.477,149.016
C07283=1209.325,-51.265,-40.129,179.808,5.476,149.017
C07284=1209.331,-51.515,-40.117,179.805,5.475,149.017
C07285=1209.336,-51.765,-40.105,179.803,5.476,149.018
C07286=1209.341,-52.014,-40.093,179.800,5.475,149.019
C07287=1209.346,-52.264,-40.081,179.798,5.476,149.020
C07288=1209.352,-52.514,-40.069,179.796,5.475,149.020
C07289=1209.357,-52.763,-40.057,179.793,5.475,149.021
C07290=1209.362,-53.013,-40.045,179.791,5.475,149.022
C07291=1209.367,-53.263,-40.033,179.788,5.475,149.022
C07292=1209.372,-53.512,-40.021,179.786,5.474,149.023
C07293=1209.377,-53.762,-40.009,179.784,5.474,149.024
C07294=1209.382,-54.012,-39.998,179.781,5.474,149.024
C07295=1209.387,-54.262,-39.986,179.779,5.474,149.025
C07296=1209.393,-54.511,-39.973,179.777,5.474,149.026
C07297=1209.398,-54.761,-39.961,179.774,5.473,149.026
C07298=1209.403,-55.010,-39.950,179.772,5.473,149.027
C07299=1209.408,-55.260,-39.938,179.769,5.473,149.028
